LIN {X 0,Y 553.099,Z 303.445,A -85,B 0,C 180,E1 26748.452,E2 26748.452} C_VEL
LIN {X 0,Y 552.954,Z 317.128,A -85,B 0,C 180,E1 26747.901,E2 26747.901} C_VEL
LIN {X 0,Y 552.726,Z 331.261,A -85,B 0,C 180,E1 26747.108,E2 26747.108} C_VEL
LIN {X 0,Y 552.512,Z 344.277,A -85,B 0,C 180,E1 26746.127,E2 26746.127} C_VEL
LIN {X 0,Y 552.313,Z 355.732,A -85,B 0,C 180,E1 26745.002,E2 26745.002} C_VEL
LIN {X 0,Y 552.151,Z 365.084,A -85,B 0,C 180,E1 26743.828,E2 26743.828} C_VEL
LIN {X 0,Y 552.032,Z 373.305,A -85,B 0,C 180,E1 26742.509,E2 26742.509} C_VEL
LIN {X 0,Y 551.958,Z 380.058,A -85,B 0,C 180,E1 26741.069,E2 26741.069} C_VEL
LIN {X 0,Y 551.926,Z 385.3,A -85,B 0,C 180,E1 26739.488,E2 26739.488} C_VEL
LIN {X 0,Y 551.919,Z 388.545,A -85,B 0,C 180,E1 26737.913,E2 26737.913} C_VEL
LIN {X 0,Y 551.917,Z 389.9,A -85,B 0,C 180,E1 26736.448,E2 26736.448} C_VEL
LIN {X 0,Y 551.917,Z 389.555,A -85,B 0,C 180,E1 26734.868,E2 26734.868} C_VEL
LIN {X 0,Y 551.918,Z 387.388,A -85,B 0,C 180,E1 26733.323,E2 26733.323} C_VEL
LIN {X 0,Y 551.933,Z 383.684,A -85,B 0,C 180,E1 26731.868,E2 26731.868} C_VEL
LIN {X 0,Y 551.979,Z 377.809,A -85,B 0,C 180,E1 26730.311,E2 26730.311} C_VEL
LIN {X 0,Y 552.075,Z 370.189,A -85,B 0,C 180,E1 26728.858,E2 26728.858} C_VEL
LIN {X 0,Y 552.222,Z 360.795,A -85,B 0,C 180,E1 26727.509,E2 26727.509} C_VEL
LIN {X 0,Y 552.402,Z 350.546,A -85,B 0,C 180,E1 26726.367,E2 26726.367} C_VEL
LIN {X 0,Y 552.574,Z 339.331,A -85,B 0,C 180,E1 26725.381,E2 26725.381} C_VEL
LIN {X 0,Y 552.815,Z 326.337,A -85,B 0,C 180,E1 26724.499,E2 26724.499} C_VEL
LIN {X 0,Y 552.997,Z 311.82,A -85,B 0,C 180,E1 26723.771,E2 26723.771} C_VEL
LIN {X 0,Y 553.096,Z 297.074,A -85,B 0,C 180,E1 26723.264,E2 26723.264} C_VEL
LIN {X 0,Y 553.162,Z 282.134,A -85,B 0,C 180,E1 26722.957,E2 26722.957} C_VEL
LIN {X 0,Y 553.318,Z 174.705,A -85,B 0,C 180,E1 26721.544,E2 26721.544} C_VEL
LIN {X 0,Y 553.702,Z 126.564,A -85,B 0,C 180,E1 26718.489,E2 26718.489} C_VEL
LIN {X 0,Y 554.116,Z 77.408,A -85,B 0,C 180,E1 26715.367,E2 26715.367} C_VEL
LIN {X 0,Y 554.166,Z 60.38,A -85,B 0,C 180,E1 26714.297,E2 26714.297} C_VEL
LIN {X 0,Y 552.386,Z 53.332,A -85,B 0,C 180,E1 26713.76,E2 26713.76} C_VEL
LIN {X 0,Y 552.341,Z 52.999,A -85,B 0,C 180,E1 26713.258,E2 26713.258} C_VEL
LIN {X 0,Y 552.362,Z 53.27,A -85,B 0,C 180,E1 26712.594,E2 26712.594} C_VEL
LIN {X 0,Y 554.241,Z 59.463,A -85,B 0,C 180,E1 26712.031,E2 26712.031} C_VEL
LIN {X 0,Y 555.025,Z 62.5,A -85,B 0,C 180,E1 26711.786,E2 26711.786} C_VEL
LIN {X 0,Y 554.132,Z 113.525,A -85,B 0,C 180,E1 26708.362,E2 26708.362} C_VEL
LIN {X 0,Y 553.365,Z 164.5,A -85,B 0,C 180,E1 26704.988,E2 26704.988} C_VEL
LIN {X 0,Y 553.381,Z 172.893,A -85,B 0,C 180,E1 26704.473,E2 26704.473} C_VEL
LIN {X 0,Y 553.711,Z 182.776,A -85,B 0,C 180,E1 26704.321,E2 26704.321} C_VEL
LIN {X 0,Y 553.297,Z 287.575,A -85,B 0,C 180,E1 26702.905,E2 26702.905} C_VEL
LIN {X 0,Y 553.196,Z 302.101,A -85,B 0,C 180,E1 26702.529,E2 26702.529} C_VEL
LIN {X 0,Y 553.009,Z 316.307,A -85,B 0,C 180,E1 26701.96,E2 26701.96} C_VEL
LIN {X 0,Y 552.788,Z 329.378,A -85,B 0,C 180,E1 26701.241,E2 26701.241} C_VEL
LIN {X 0,Y 552.561,Z 342.406,A -85,B 0,C 180,E1 26700.293,E2 26700.293} C_VEL
LIN {X 0,Y 552.346,Z 354.092,A -85,B 0,C 180,E1 26699.183,E2 26699.183} C_VEL
LIN {X 0,Y 552.173,Z 363.791,A -85,B 0,C 180,E1 26698.009,E2 26698.009} C_VEL
LIN {X 0,Y 552.049,Z 372.165,A -85,B 0,C 180,E1 26696.716,E2 26696.716} C_VEL
LIN {X 0,Y 551.963,Z 379.488,A -85,B 0,C 180,E1 26695.207,E2 26695.207} C_VEL
LIN {X 0,Y 551.928,Z 384.789,A -85,B 0,C 180,E1 26693.673,E2 26693.673} C_VEL
LIN {X 0,Y 551.918,Z 388.153,A -85,B 0,C 180,E1 26692.173,E2 26692.173} C_VEL
LIN {X 0,Y 551.919,Z 389.809,A -85,B 0,C 180,E1 26690.649,E2 26690.649} C_VEL
LIN {X 0,Y 551.917,Z 389.741,A -85,B 0,C 180,E1 26689.157,E2 26689.157} C_VEL
LIN {X 0,Y 551.918,Z 387.985,A -85,B 0,C 180,E1 26687.63,E2 26687.63} C_VEL
LIN {X 0,Y 551.928,Z 384.27,A -85,B 0,C 180,E1 26686.066,E2 26686.066} C_VEL
LIN {X 0,Y 551.969,Z 379.118,A -85,B 0,C 180,E1 26684.61,E2 26684.61} C_VEL
LIN {X 0,Y 552.051,Z 372.285,A -85,B 0,C 180,E1 26683.206,E2 26683.206} C_VEL
LIN {X 0,Y 552.19,Z 363.437,A -85,B 0,C 180,E1 26681.84,E2 26681.84} C_VEL
LIN {X 0,Y 552.372,Z 353.642,A -85,B 0,C 180,E1 26680.666,E2 26680.666} C_VEL
LIN {X 0,Y 552.577,Z 342.861,A -85,B 0,C 180,E1 26679.641,E2 26679.641} C_VEL
LIN {X 0,Y 552.83,Z 329.763,A -85,B 0,C 180,E1 26678.678,E2 26678.678} C_VEL
LIN {X 0,Y 553.049,Z 316.225,A -85,B 0,C 180,E1 26677.93,E2 26677.93} C_VEL
LIN {X 0,Y 553.237,Z 302.018,A -85,B 0,C 180,E1 26677.362,E2 26677.362} C_VEL
LIN {X 0,Y 553.37,Z 286.424,A -85,B 0,C 180,E1 26676.965,E2 26676.965} C_VEL
LIN {X 0,Y 553.62,Z 179.911,A -85,B 0,C 180,E1 26675.504,E2 26675.504} C_VEL
LIN {X 0,Y 552.92,Z 175.405,A -85,B 0,C 180,E1 26675.389,E2 26675.389} C_VEL
LIN {X 0,Y 553.371,Z 145.57,A -85,B 0,C 180,E1 26672.069,E2 26672.069} C_VEL
LIN {X 0,Y 554.026,Z 115.936,A -85,B 0,C 180,E1 26668.707,E2 26668.707} C_VEL
LIN {X 0,Y 554.696,Z 87.232,A -85,B 0,C 180,E1 26665.405,E2 26665.405} C_VEL
LIN {X 0,Y 555.219,Z 63.854,A -85,B 0,C 180,E1 26662.668,E2 26662.668} C_VEL
LIN {X 0,Y 552.318,Z 53.131,A -85,B 0,C 180,E1 26661.162,E2 26661.162} C_VEL
LIN {X 0,Y 552.344,Z 52.997,A -85,B 0,C 180,E1 26657.923,E2 26657.923} C_VEL
LIN {X 0,Y 552.305,Z 52.997,A -85,B 0,C 180,E1 26654.682,E2 26654.682} C_VEL
LIN {X 0,Y 552.297,Z 52.998,A -85,B 0,C 180,E1 26651.381,E2 26651.381} C_VEL
LIN {X 0,Y 552.344,Z 52.997,A -85,B 0,C 180,E1 26648.117,E2 26648.117} C_VEL
LIN {X 0,Y 552.298,Z 52.998,A -85,B 0,C 180,E1 26644.881,E2 26644.881} C_VEL
LIN {X 0,Y 552.291,Z 52.998,A -85,B 0,C 180,E1 26641.556,E2 26641.556} C_VEL
LIN {X 0,Y 552.345,Z 52.999,A -85,B 0,C 180,E1 26638.341,E2 26638.341} C_VEL
LIN {X 0,Y 552.292,Z 52.998,A -85,B 0,C 180,E1 26635.119,E2 26635.119} C_VEL
LIN {X 0,Y 552.287,Z 52.999,A -85,B 0,C 180,E1 26631.777,E2 26631.777} C_VEL
LIN {X 0,Y 552.34,Z 52.999,A -85,B 0,C 180,E1 26628.514,E2 26628.514} C_VEL
LIN {X 0,Y 552.286,Z 52.998,A -85,B 0,C 180,E1 26625.318,E2 26625.318} C_VEL
LIN {X 0,Y 552.28,Z 52.998,A -85,B 0,C 180,E1 26621.966,E2 26621.966} C_VEL
LIN {X 0,Y 552.342,Z 52.998,A -85,B 0,C 180,E1 26618.774,E2 26618.774} C_VEL
LIN {X 0,Y 552.277,Z 52.999,A -85,B 0,C 180,E1 26615.594,E2 26615.594} C_VEL
LIN {X 0,Y 552.276,Z 53,A -85,B 0,C 180,E1 26612.154,E2 26612.154} C_VEL
LIN {X 0,Y 552.334,Z 53,A -85,B 0,C 180,E1 26608.941,E2 26608.941} C_VEL
LIN {X 0,Y 552.279,Z 53,A -85,B 0,C 180,E1 26605.645,E2 26605.645} C_VEL
LIN {X 0,Y 552.266,Z 53.001,A -85,B 0,C 180,E1 26602.27,E2 26602.27} C_VEL
LIN {X 0,Y 552.323,Z 53.002,A -85,B 0,C 180,E1 26599.056,E2 26599.056} C_VEL
LIN {X 0,Y 552.278,Z 53,A -85,B 0,C 180,E1 26595.812,E2 26595.812} C_VEL
LIN {X 0,Y 552.267,Z 53.002,A -85,B 0,C 180,E1 26592.478,E2 26592.478} C_VEL
LIN {X 0,Y 552.337,Z 52.998,A -85,B 0,C 180,E1 26589.315,E2 26589.315} C_VEL
LIN {X 0,Y 552.282,Z 53.003,A -85,B 0,C 180,E1 26586.043,E2 26586.043} C_VEL
LIN {X 0,Y 552.272,Z 52.996,A -85,B 0,C 180,E1 26582.663,E2 26582.663} C_VEL
LIN {X 0,Y 552.347,Z 53.475,A -85,B 0,C 180,E1 26582.323,E2 26582.323} C_VEL
LIN {X 0,Y 556.547,Z 66.471,A -85,B 0,C 180,E1 26581.038,E2 26581.038} C_VEL
LIN {X 0,Y 555.743,Z 104.341,A -85,B 0,C 180,E1 26578.241,E2 26578.241} C_VEL
LIN {X 0,Y 554.952,Z 151.652,A -85,B 0,C 180,E1 26574.86,E2 26574.86} C_VEL
LIN {X 0,Y 554.938,Z 158.626,A -85,B 0,C 180,E1 26574.402,E2 26574.402} C_VEL
LIN {X 0,Y 555.863,Z 167.052,A -85,B 0,C 180,E1 26574.255,E2 26574.255} C_VEL
LIN {X 0,Y 555.252,Z 366.942,A -85,B 0,C 180,E1 26571.605,E2 26571.605} C_VEL
LIN {X 0,Y 555.016,Z 386.194,A -85,B 0,C 180,E1 26571.154,E2 26571.154} C_VEL
LIN {X 0,Y 554.725,Z 404.372,A -85,B 0,C 180,E1 26570.539,E2 26570.539} C_VEL
LIN {X 0,Y 554.4,Z 421.777,A -85,B 0,C 180,E1 26569.765,E2 26569.765} C_VEL
LIN {X 0,Y 554.022,Z 437.939,A -85,B 0,C 180,E1 26568.848,E2 26568.848} C_VEL
LIN {X 0,Y 553.586,Z 454.217,A -85,B 0,C 180,E1 26567.697,E2 26567.697} C_VEL
LIN {X 0,Y 553.179,Z 468.99,A -85,B 0,C 180,E1 26566.432,E2 26566.432} C_VEL
LIN {X 0,Y 552.81,Z 483.013,A -85,B 0,C 180,E1 26564.99,E2 26564.99} C_VEL
LIN {X 0,Y 552.503,Z 495.909,A -85,B 0,C 180,E1 26563.394,E2 26563.394} C_VEL
LIN {X 0,Y 552.262,Z 507.225,A -85,B 0,C 180,E1 26561.7,E2 26561.7} C_VEL
LIN {X 0,Y 552.098,Z 517.163,A -85,B 0,C 180,E1 26559.872,E2 26559.872} C_VEL
LIN {X 0,Y 551.994,Z 525.176,A -85,B 0,C 180,E1 26558.018,E2 26558.018} C_VEL
LIN {X 0,Y 551.941,Z 531.413,A -85,B 0,C 180,E1 26556.136,E2 26556.136} C_VEL
LIN {X 0,Y 551.914,Z 535.875,A -85,B 0,C 180,E1 26554.26,E2 26554.26} C_VEL
LIN {X 0,Y 551.913,Z 538.792,A -85,B 0,C 180,E1 26552.285,E2 26552.285} C_VEL
LIN {X 0,Y 551.908,Z 539.939,A -85,B 0,C 180,E1 26550.312,E2 26550.312} C_VEL
LIN {X 0,Y 551.913,Z 539.415,A -85,B 0,C 180,E1 26548.444,E2 26548.444} C_VEL
LIN {X 0,Y 551.91,Z 537.163,A -85,B 0,C 180,E1 26546.469,E2 26546.469} C_VEL
LIN {X 0,Y 551.929,Z 533.352,A -85,B 0,C 180,E1 26544.596,E2 26544.596} C_VEL
LIN {X 0,Y 551.964,Z 527.822,A -85,B 0,C 180,E1 26542.716,E2 26542.716} C_VEL
LIN {X 0,Y 552.054,Z 520.43,A -85,B 0,C 180,E1 26540.83,E2 26540.83} C_VEL
LIN {X 0,Y 552.185,Z 511.522,A -85,B 0,C 180,E1 26539.041,E2 26539.041} C_VEL
LIN {X 0,Y 552.389,Z 500.984,A -85,B 0,C 180,E1 26537.323,E2 26537.323} C_VEL
LIN {X 0,Y 552.655,Z 489.359,A -85,B 0,C 180,E1 26535.757,E2 26535.757} C_VEL
LIN {X 0,Y 552.991,Z 476.089,A -85,B 0,C 180,E1 26534.265,E2 26534.265} C_VEL
LIN {X 0,Y 553.394,Z 461.229,A -85,B 0,C 180,E1 26532.873,E2 26532.873} C_VEL
LIN {X 0,Y 553.836,Z 445.249,A -85,B 0,C 180,E1 26531.638,E2 26531.638} C_VEL
LIN {X 0,Y 554.249,Z 428.995,A -85,B 0,C 180,E1 26530.615,E2 26530.615} C_VEL
LIN {X 0,Y 554.606,Z 411.48,A -85,B 0,C 180,E1 26529.75,E2 26529.75} C_VEL
LIN {X 0,Y 554.93,Z 392.522,A -85,B 0,C 180,E1 26529.035,E2 26529.035} C_VEL
LIN {X 0,Y 555.188,Z 373.634,A -85,B 0,C 180,E1 26528.526,E2 26528.526} C_VEL
LIN {X 0,Y 555.342,Z 353.291,A -85,B 0,C 180,E1 26528.186,E2 26528.186} C_VEL
LIN {X 0,Y 555.788,Z 158.707,A -85,B 0,C 180,E1 26525.612,E2 26525.612} C_VEL
LIN {X 0,Y 555.53,Z 154.307,A -85,B 0,C 180,E1 26525.516,E2 26525.516} C_VEL
LIN {X 0,Y 556.369,Z 79.517,A -85,B 0,C 180,E1 26522.378,E2 26522.378} C_VEL
LIN {X 0,Y 556.405,Z 64.239,A -85,B 0,C 180,E1 26521.706,E2 26521.706} C_VEL
LIN {X 0,Y 552.416,Z 53.549,A -85,B 0,C 180,E1 26520.999,E2 26520.999} C_VEL
LIN {X 0,Y 552.331,Z 52.991,A -85,B 0,C 180,E1 26520.755,E2 26520.755} C_VEL
LIN {X 0,Y 552.33,Z 52.994,A -85,B 0,C 180,E1 26517.327,E2 26517.327} C_VEL
LIN {X 0,Y 552.333,Z 52.997,A -85,B 0,C 180,E1 26513.963,E2 26513.963} C_VEL
LIN {X 0,Y 552.342,Z 52.992,A -85,B 0,C 180,E1 26510.553,E2 26510.553} C_VEL
LIN {X 0,Y 552.324,Z 52.995,A -85,B 0,C 180,E1 26507.248,E2 26507.248} C_VEL
LIN {X 0,Y 552.341,Z 52.998,A -85,B 0,C 180,E1 26503.893,E2 26503.893} C_VEL
LIN {X 0,Y 552.336,Z 52.993,A -85,B 0,C 180,E1 26500.512,E2 26500.512} C_VEL
LIN {X 0,Y 552.325,Z 52.993,A -85,B 0,C 180,E1 26497.202,E2 26497.202} C_VEL
LIN {X 0,Y 552.322,Z 52.997,A -85,B 0,C 180,E1 26493.763,E2 26493.763} C_VEL
LIN {X 0,Y 552.339,Z 52.995,A -85,B 0,C 180,E1 26490.455,E2 26490.455} C_VEL
LIN {X 0,Y 552.34,Z 52.99,A -85,B 0,C 180,E1 26487.024,E2 26487.024} C_VEL
LIN {X 0,Y 552.314,Z 52.992,A -85,B 0,C 180,E1 26483.654,E2 26483.654} C_VEL
LIN {X 0,Y 552.335,Z 52.997,A -85,B 0,C 180,E1 26480.335,E2 26480.335} C_VEL
LIN {X 0,Y 552.341,Z 52.994,A -85,B 0,C 180,E1 26476.944,E2 26476.944} C_VEL
LIN {X 0,Y 552.319,Z 52.992,A -85,B 0,C 180,E1 26473.611,E2 26473.611} C_VEL
LIN {X 0,Y 552.313,Z 52.994,A -85,B 0,C 180,E1 26470.219,E2 26470.219} C_VEL
LIN {X 0,Y 552.343,Z 52.998,A -85,B 0,C 180,E1 26466.862,E2 26466.862} C_VEL
LIN {X 0,Y 552.339,Z 52.991,A -85,B 0,C 180,E1 26463.425,E2 26463.425} C_VEL
LIN {X 0,Y 552.306,Z 52.992,A -85,B 0,C 180,E1 26460.104,E2 26460.104} C_VEL
LIN {X 0,Y 552.323,Z 52.998,A -85,B 0,C 180,E1 26456.762,E2 26456.762} C_VEL
LIN {X 0,Y 552.344,Z 52.993,A -85,B 0,C 180,E1 26453.451,E2 26453.451} C_VEL
LIN {X 0,Y 552.304,Z 52.993,A -85,B 0,C 180,E1 26450.202,E2 26450.202} C_VEL
LIN {X 0,Y 552.31,Z 52.995,A -85,B 0,C 180,E1 26446.814,E2 26446.814} C_VEL
LIN {X 0,Y 552.344,Z 52.997,A -85,B 0,C 180,E1 26443.489,E2 26443.489} C_VEL
LIN {X 0,Y 552.31,Z 52.995,A -85,B 0,C 180,E1 26440.212,E2 26440.212} C_VEL
LIN {X 0,Y 552.298,Z 52.989,A -85,B 0,C 180,E1 26436.868,E2 26436.868} C_VEL
LIN {X 0,Y 552.341,Z 52.998,A -85,B 0,C 180,E1 26433.556,E2 26433.556} C_VEL
LIN {X 0,Y 552.294,Z 52.997,A -85,B 0,C 180,E1 26432.704,E2 26432.704} C_VEL
LIN {X 0,Y 551.318,Z 53.124,A -85,B 0,C 180,E1 26431.905,E2 26431.905} C_VEL
LIN {X 0,Y 544.811,Z 53.932,A -85,B 0,C 180,E1 26429.603,E2 26429.603} C_VEL
LIN {X 0,Y 544.359,Z 53.984,A -85,B 0,C 180,E1 26429.076,E2 26429.076} C_VEL
LIN {X 0,Y 544.403,Z 53.986,A -85,B 0,C 180,E1 26425.736,E2 26425.736} C_VEL
LIN {X 0,Y 544.373,Z 53.985,A -85,B 0,C 180,E1 26422.425,E2 26422.425} C_VEL
LIN {X 0,Y 544.352,Z 53.986,A -85,B 0,C 180,E1 26419.164,E2 26419.164} C_VEL
LIN {X 0,Y 544.395,Z 53.985,A -85,B 0,C 180,E1 26415.886,E2 26415.886} C_VEL
LIN {X 0,Y 544.364,Z 53.983,A -85,B 0,C 180,E1 26412.667,E2 26412.667} C_VEL
LIN {X 0,Y 544.344,Z 53.99,A -85,B 0,C 180,E1 26409.322,E2 26409.322} C_VEL
LIN {X 0,Y 544.391,Z 53.989,A -85,B 0,C 180,E1 26406.086,E2 26406.086} C_VEL
LIN {X 0,Y 544.387,Z 54.212,A -85,B 0,C 180,E1 26403.766,E2 26403.766} C_VEL
LIN {X 0,Y 545.826,Z 61.376,A -85,B 0,C 180,E1 26402.958,E2 26402.958} C_VEL
LIN {X 0,Y 545.926,Z 92.268,A -85,B 0,C 180,E1 26399.756,E2 26399.756} C_VEL
LIN {X 0,Y 545.776,Z 123.082,A -85,B 0,C 180,E1 26396.489,E2 26396.489} C_VEL
LIN {X 0,Y 545.516,Z 153.208,A -85,B 0,C 180,E1 26393.264,E2 26393.264} C_VEL
LIN {X 0,Y 545.269,Z 178.791,A -85,B 0,C 180,E1 26390.544,E2 26390.544} C_VEL
LIN {X 0,Y 545.789,Z 185.113,A -85,B 0,C 180,E1 26390.438,E2 26390.438} C_VEL
LIN {X 0,Y 545.419,Z 289.991,A -85,B 0,C 180,E1 26389.023,E2 26389.023} C_VEL
LIN {X 0,Y 545.341,Z 304.564,A -85,B 0,C 180,E1 26388.63,E2 26388.63} C_VEL
LIN {X 0,Y 545.187,Z 318.586,A -85,B 0,C 180,E1 26388.055,E2 26388.055} C_VEL
LIN {X 0,Y 544.956,Z 332.024,A -85,B 0,C 180,E1 26387.29,E2 26387.29} C_VEL
LIN {X 0,Y 544.717,Z 344.949,A -85,B 0,C 180,E1 26386.309,E2 26386.309} C_VEL
LIN {X 0,Y 544.502,Z 356.015,A -85,B 0,C 180,E1 26385.223,E2 26385.223} C_VEL
LIN {X 0,Y 544.314,Z 365.564,A -85,B 0,C 180,E1 26384.031,E2 26384.031} C_VEL
LIN {X 0,Y 544.159,Z 374.274,A -85,B 0,C 180,E1 26382.629,E2 26382.629} C_VEL
LIN {X 0,Y 544.062,Z 381.231,A -85,B 0,C 180,E1 26381.125,E2 26381.125} C_VEL
LIN {X 0,Y 544.009,Z 386.403,A -85,B 0,C 180,E1 26379.52,E2 26379.52} C_VEL
LIN {X 0,Y 543.982,Z 389.541,A -85,B 0,C 180,E1 26377.923,E2 26377.923} C_VEL
LIN {X 0,Y 543.971,Z 390.853,A -85,B 0,C 180,E1 26376.331,E2 26376.331} C_VEL
LIN {X 0,Y 543.973,Z 390.407,A -85,B 0,C 180,E1 26374.744,E2 26374.744} C_VEL
LIN {X 0,Y 543.991,Z 387.95,A -85,B 0,C 180,E1 26373.055,E2 26373.055} C_VEL
LIN {X 0,Y 544.033,Z 383.689,A -85,B 0,C 180,E1 26371.474,E2 26371.474} C_VEL
LIN {X 0,Y 544.102,Z 377.829,A -85,B 0,C 180,E1 26369.999,E2 26369.999} C_VEL
LIN {X 0,Y 544.219,Z 370.506,A -85,B 0,C 180,E1 26368.631,E2 26368.631} C_VEL
LIN {X 0,Y 544.385,Z 361.73,A -85,B 0,C 180,E1 26367.367,E2 26367.367} C_VEL
LIN {X 0,Y 544.591,Z 351.43,A -85,B 0,C 180,E1 26366.21,E2 26366.21} C_VEL
LIN {X 0,Y 544.785,Z 340.151,A -85,B 0,C 180,E1 26365.209,E2 26365.209} C_VEL
LIN {X 0,Y 545.047,Z 327.077,A -85,B 0,C 180,E1 26364.314,E2 26364.314} C_VEL
LIN {X 0,Y 545.241,Z 312.435,A -85,B 0,C 180,E1 26363.577,E2 26363.577} C_VEL
LIN {X 0,Y 545.348,Z 296.996,A -85,B 0,C 180,E1 26363.049,E2 26363.049} C_VEL
LIN {X 0,Y 545.398,Z 281.169,A -85,B 0,C 180,E1 26362.742,E2 26362.742} C_VEL
LIN {X 0,Y 545.609,Z 175.423,A -85,B 0,C 180,E1 26361.33,E2 26361.33} C_VEL
LIN {X 0,Y 546.063,Z 123.971,A -85,B 0,C 180,E1 26358.058,E2 26358.058} C_VEL
LIN {X 0,Y 546.484,Z 71.6,A -85,B 0,C 180,E1 26354.724,E2 26354.724} C_VEL
LIN {X 0,Y 546.407,Z 61.981,A -85,B 0,C 180,E1 26354.123,E2 26354.123} C_VEL
LIN {X 0,Y 544.455,Z 54.321,A -85,B 0,C 180,E1 26353.53,E2 26353.53} C_VEL
LIN {X 0,Y 544.396,Z 53.991,A -85,B 0,C 180,E1 26353.116,E2 26353.116} C_VEL
LIN {X 0,Y 544.488,Z 54.61,A -85,B 0,C 180,E1 26352.858,E2 26352.858} C_VEL
LIN {X 0,Y 547.518,Z 64.97,A -85,B 0,C 180,E1 26351.968,E2 26351.968} C_VEL
LIN {X 0,Y 546.527,Z 115.573,A -85,B 0,C 180,E1 26348.537,E2 26348.537} C_VEL
LIN {X 0,Y 545.66,Z 166.93,A -85,B 0,C 180,E1 26345.099,E2 26345.099} C_VEL
LIN {X 0,Y 545.704,Z 172.937,A -85,B 0,C 180,E1 26344.742,E2 26344.742} C_VEL
LIN {X 0,Y 546.13,Z 181.831,A -85,B 0,C 180,E1 26344.6,E2 26344.6} C_VEL
LIN {X 0,Y 545.622,Z 288.062,A -85,B 0,C 180,E1 26343.135,E2 26343.135} C_VEL
LIN {X 0,Y 545.499,Z 303.41,A -85,B 0,C 180,E1 26342.727,E2 26342.727} C_VEL
LIN {X 0,Y 545.278,Z 318.268,A -85,B 0,C 180,E1 26342.109,E2 26342.109} C_VEL
LIN {X 0,Y 545.031,Z 330.81,A -85,B 0,C 180,E1 26341.392,E2 26341.392} C_VEL
LIN {X 0,Y 544.781,Z 343.449,A -85,B 0,C 180,E1 26340.454,E2 26340.454} C_VEL
LIN {X 0,Y 544.529,Z 355.341,A -85,B 0,C 180,E1 26339.305,E2 26339.305} C_VEL
LIN {X 0,Y 544.324,Z 365.014,A -85,B 0,C 180,E1 26338.108,E2 26338.108} C_VEL
LIN {X 0,Y 544.175,Z 373.324,A -85,B 0,C 180,E1 26336.801,E2 26336.801} C_VEL
LIN {X 0,Y 544.066,Z 380.786,A -85,B 0,C 180,E1 26335.233,E2 26335.233} C_VEL
LIN {X 0,Y 544.01,Z 386.15,A -85,B 0,C 180,E1 26333.613,E2 26333.613} C_VEL
LIN {X 0,Y 543.982,Z 389.363,A -85,B 0,C 180,E1 26332.048,E2 26332.048} C_VEL
LIN {X 0,Y 543.973,Z 390.829,A -85,B 0,C 180,E1 26330.508,E2 26330.508} C_VEL
LIN {X 0,Y 543.975,Z 390.517,A -85,B 0,C 180,E1 26328.85,E2 26328.85} C_VEL
LIN {X 0,Y 543.995,Z 388.455,A -85,B 0,C 180,E1 26327.295,E2 26327.295} C_VEL
LIN {X 0,Y 544.035,Z 384.784,A -85,B 0,C 180,E1 26325.788,E2 26325.788} C_VEL
LIN {X 0,Y 544.105,Z 378.968,A -85,B 0,C 180,E1 26324.22,E2 26324.22} C_VEL
LIN {X 0,Y 544.222,Z 371.846,A -85,B 0,C 180,E1 26322.826,E2 26322.826} C_VEL
LIN {X 0,Y 544.398,Z 363.265,A -85,B 0,C 180,E1 26321.531,E2 26321.531} C_VEL
LIN {X 0,Y 544.642,Z 352.354,A -85,B 0,C 180,E1 26320.257,E2 26320.257} C_VEL
LIN {X 0,Y 544.89,Z 340.946,A -85,B 0,C 180,E1 26319.222,E2 26319.222} C_VEL
LIN {X 0,Y 545.16,Z 328.543,A -85,B 0,C 180,E1 26318.343,E2 26318.343} C_VEL
LIN {X 0,Y 545.405,Z 315.197,A -85,B 0,C 180,E1 26317.624,E2 26317.624} C_VEL
LIN {X 0,Y 545.601,Z 300.554,A -85,B 0,C 180,E1 26317.062,E2 26317.062} C_VEL
LIN {X 0,Y 545.735,Z 285.71,A -85,B 0,C 180,E1 26316.702,E2 26316.702} C_VEL
LIN {X 0,Y 546.094,Z 180.817,A -85,B 0,C 180,E1 26315.23,E2 26315.23} C_VEL
LIN {X 0,Y 545.172,Z 175.182,A -85,B 0,C 180,E1 26315.082,E2 26315.082} C_VEL
LIN {X 0,Y 545.69,Z 145.44,A -85,B 0,C 180,E1 26311.727,E2 26311.727} C_VEL
LIN {X 0,Y 546.426,Z 115.516,A -85,B 0,C 180,E1 26308.29,E2 26308.29} C_VEL
LIN {X 0,Y 547.207,Z 87.033,A -85,B 0,C 180,E1 26304.967,E2 26304.967} C_VEL
LIN {X 0,Y 547.749,Z 66.487,A -85,B 0,C 180,E1 26302.535,E2 26302.535} C_VEL
LIN {X 0,Y 544.375,Z 54.101,A -85,B 0,C 180,E1 26300.762,E2 26300.762} C_VEL
LIN {X 0,Y 544.369,Z 53.99,A -85,B 0,C 180,E1 26297.421,E2 26297.421} C_VEL
LIN {X 0,Y 544.409,Z 53.986,A -85,B 0,C 180,E1 26294.136,E2 26294.136} C_VEL
LIN {X 0,Y 544.356,Z 53.986,A -85,B 0,C 180,E1 26290.906,E2 26290.906} C_VEL
LIN {X 0,Y 544.356,Z 53.988,A -85,B 0,C 180,E1 26287.494,E2 26287.494} C_VEL
LIN {X 0,Y 544.404,Z 53.988,A -85,B 0,C 180,E1 26284.213,E2 26284.213} C_VEL
LIN {X 0,Y 544.36,Z 53.986,A -85,B 0,C 180,E1 26280.947,E2 26280.947} C_VEL
LIN {X 0,Y 544.347,Z 53.988,A -85,B 0,C 180,E1 26277.579,E2 26277.579} C_VEL
LIN {X 0,Y 544.397,Z 53.988,A -85,B 0,C 180,E1 26274.308,E2 26274.308} C_VEL
LIN {X 0,Y 544.357,Z 53.987,A -85,B 0,C 180,E1 26271.125,E2 26271.125} C_VEL
LIN {X 0,Y 544.343,Z 53.988,A -85,B 0,C 180,E1 26267.737,E2 26267.737} C_VEL
LIN {X 0,Y 544.386,Z 53.988,A -85,B 0,C 180,E1 26264.446,E2 26264.446} C_VEL
LIN {X 0,Y 544.355,Z 53.986,A -85,B 0,C 180,E1 26261.25,E2 26261.25} C_VEL
LIN {X 0,Y 544.337,Z 53.988,A -85,B 0,C 180,E1 26257.993,E2 26257.993} C_VEL
LIN {X 0,Y 544.394,Z 53.989,A -85,B 0,C 180,E1 26254.78,E2 26254.78} C_VEL
LIN {X 0,Y 544.341,Z 53.989,A -85,B 0,C 180,E1 26251.593,E2 26251.593} C_VEL
LIN {X 0,Y 544.331,Z 53.99,A -85,B 0,C 180,E1 26248.185,E2 26248.185} C_VEL
LIN {X 0,Y 544.383,Z 53.99,A -85,B 0,C 180,E1 26244.909,E2 26244.909} C_VEL
LIN {X 0,Y 544.342,Z 53.99,A -85,B 0,C 180,E1 26241.658,E2 26241.658} C_VEL
LIN {X 0,Y 544.324,Z 53.991,A -85,B 0,C 180,E1 26238.322,E2 26238.322} C_VEL
LIN {X 0,Y 544.386,Z 53.989,A -85,B 0,C 180,E1 26235.148,E2 26235.148} C_VEL
LIN {X 0,Y 544.34,Z 53.991,A -85,B 0,C 180,E1 26231.934,E2 26231.934} C_VEL
LIN {X 0,Y 544.334,Z 53.992,A -85,B 0,C 180,E1 26228.648,E2 26228.648} C_VEL
LIN {X 0,Y 544.392,Z 53.989,A -85,B 0,C 180,E1 26225.366,E2 26225.366} C_VEL
LIN {X 0,Y 544.376,Z 54.248,A -85,B 0,C 180,E1 26222.777,E2 26222.777} C_VEL
LIN {X 0,Y 549.194,Z 68.607,A -85,B 0,C 180,E1 26221.293,E2 26221.293} C_VEL
LIN {X 0,Y 548.134,Z 110.619,A -85,B 0,C 180,E1 26218.134,E2 26218.134} C_VEL
LIN {X 0,Y 547.224,Z 157.206,A -85,B 0,C 180,E1 26214.757,E2 26214.757} C_VEL
LIN {X 0,Y 547.437,Z 159.937,A -85,B 0,C 180,E1 26214.657,E2 26214.657} C_VEL
LIN {X 0,Y 548.298,Z 168.095,A -85,B 0,C 180,E1 26214.515,E2 26214.515} C_VEL
LIN {X 0,Y 547.592,Z 366.306,A -85,B 0,C 180,E1 26211.855,E2 26211.855} C_VEL
LIN {X 0,Y 547.319,Z 385.448,A -85,B 0,C 180,E1 26211.402,E2 26211.402} C_VEL
LIN {X 0,Y 546.977,Z 403.863,A -85,B 0,C 180,E1 26210.771,E2 26210.771} C_VEL
LIN {X 0,Y 546.58,Z 422.045,A -85,B 0,C 180,E1 26209.943,E2 26209.943} C_VEL
LIN {X 0,Y 546.163,Z 439.093,A -85,B 0,C 180,E1 26208.963,E2 26208.963} C_VEL
LIN {X 0,Y 545.743,Z 455.363,A -85,B 0,C 180,E1 26207.817,E2 26207.817} C_VEL
LIN {X 0,Y 545.352,Z 470.045,A -85,B 0,C 180,E1 26206.565,E2 26206.565} C_VEL
LIN {X 0,Y 544.957,Z 483.221,A -85,B 0,C 180,E1 26205.187,E2 26205.187} C_VEL
LIN {X 0,Y 544.604,Z 495.908,A -85,B 0,C 180,E1 26203.592,E2 26203.592} C_VEL
LIN {X 0,Y 544.327,Z 507.224,A -85,B 0,C 180,E1 26201.873,E2 26201.873} C_VEL
LIN {X 0,Y 544.133,Z 516.989,A -85,B 0,C 180,E1 26200.054,E2 26200.054} C_VEL
LIN {X 0,Y 544.007,Z 525.175,A -85,B 0,C 180,E1 26198.137,E2 26198.137} C_VEL
LIN {X 0,Y 543.944,Z 531.413,A -85,B 0,C 180,E1 26196.227,E2 26196.227} C_VEL
LIN {X 0,Y 543.916,Z 535.875,A -85,B 0,C 180,E1 26194.323,E2 26194.323} C_VEL
LIN {X 0,Y 543.912,Z 538.791,A -85,B 0,C 180,E1 26192.319,E2 26192.319} C_VEL
LIN {X 0,Y 543.908,Z 539.939,A -85,B 0,C 180,E1 26190.317,E2 26190.317} C_VEL
LIN {X 0,Y 543.912,Z 539.415,A -85,B 0,C 180,E1 26188.421,E2 26188.421} C_VEL
LIN {X 0,Y 543.911,Z 537.162,A -85,B 0,C 180,E1 26186.417,E2 26186.417} C_VEL
LIN {X 0,Y 543.931,Z 533.351,A -85,B 0,C 180,E1 26184.516,E2 26184.516} C_VEL
LIN {X 0,Y 543.976,Z 527.821,A -85,B 0,C 180,E1 26182.609,E2 26182.609} C_VEL
LIN {X 0,Y 544.076,Z 520.43,A -85,B 0,C 180,E1 26180.694,E2 26180.694} C_VEL
LIN {X 0,Y 544.236,Z 511.522,A -85,B 0,C 180,E1 26178.879,E2 26178.879} C_VEL
LIN {X 0,Y 544.467,Z 501.156,A -85,B 0,C 180,E1 26177.163,E2 26177.163} C_VEL
LIN {X 0,Y 544.783,Z 489.358,A -85,B 0,C 180,E1 26175.547,E2 26175.547} C_VEL
LIN {X 0,Y 545.177,Z 476.088,A -85,B 0,C 180,E1 26174.033,E2 26174.033} C_VEL
LIN {X 0,Y 545.549,Z 462.781,A -85,B 0,C 180,E1 26172.784,E2 26172.784} C_VEL
LIN {X 0,Y 545.973,Z 446.914,A -85,B 0,C 180,E1 26171.556,E2 26171.556} C_VEL
LIN {X 0,Y 546.404,Z 430.208,A -85,B 0,C 180,E1 26170.492,E2 26170.492} C_VEL
LIN {X 0,Y 546.805,Z 413.145,A -85,B 0,C 180,E1 26169.616,E2 26169.616} C_VEL
LIN {X 0,Y 547.176,Z 395.356,A -85,B 0,C 180,E1 26168.902,E2 26168.902} C_VEL
LIN {X 0,Y 547.488,Z 376.64,A -85,B 0,C 180,E1 26168.353,E2 26168.353} C_VEL
LIN {X 0,Y 547.698,Z 357.218,A -85,B 0,C 180,E1 26167.987,E2 26167.987} C_VEL
LIN {X 0,Y 548.265,Z 159.461,A -85,B 0,C 180,E1 26165.338,E2 26165.338} C_VEL
LIN {X 0,Y 547.969,Z 154.53,A -85,B 0,C 180,E1 26165.236,E2 26165.236} C_VEL
LIN {X 0,Y 548.899,Z 86.989,A -85,B 0,C 180,E1 26162.353,E2 26162.353} C_VEL
LIN {X 0,Y 549.159,Z 66.994,A -85,B 0,C 180,E1 26161.472,E2 26161.472} C_VEL
LIN {X 0,Y 544.495,Z 54.583,A -85,B 0,C 180,E1 26160.642,E2 26160.642} C_VEL
LIN {X 0,Y 544.41,Z 54.031,A -85,B 0,C 180,E1 26160.516,E2 26160.516} C_VEL
LIN {X 0,Y 544.387,Z 53.981,A -85,B 0,C 180,E1 26157.069,E2 26157.069} C_VEL
LIN {X 0,Y 544.4,Z 53.988,A -85,B 0,C 180,E1 26153.734,E2 26153.734} C_VEL
LIN {X 0,Y 544.394,Z 53.985,A -85,B 0,C 180,E1 26150.273,E2 26150.273} C_VEL
LIN {X 0,Y 544.395,Z 53.982,A -85,B 0,C 180,E1 26146.905,E2 26146.905} C_VEL
LIN {X 0,Y 544.385,Z 53.985,A -85,B 0,C 180,E1 26143.493,E2 26143.493} C_VEL
LIN {X 0,Y 544.401,Z 53.986,A -85,B 0,C 180,E1 26140.14,E2 26140.14} C_VEL
LIN {X 0,Y 544.399,Z 53.982,A -85,B 0,C 180,E1 26136.648,E2 26136.648} C_VEL
LIN {X 0,Y 544.385,Z 53.982,A -85,B 0,C 180,E1 26133.31,E2 26133.31} C_VEL
LIN {X 0,Y 544.383,Z 53.986,A -85,B 0,C 180,E1 26129.851,E2 26129.851} C_VEL
LIN {X 0,Y 544.4,Z 53.984,A -85,B 0,C 180,E1 26126.506,E2 26126.506} C_VEL
LIN {X 0,Y 544.404,Z 53.977,A -85,B 0,C 180,E1 26123.029,E2 26123.029} C_VEL
LIN {X 0,Y 544.375,Z 53.981,A -85,B 0,C 180,E1 26119.64,E2 26119.64} C_VEL
LIN {X 0,Y 544.382,Z 53.986,A -85,B 0,C 180,E1 26116.211,E2 26116.211} C_VEL
LIN {X 0,Y 544.401,Z 53.984,A -85,B 0,C 180,E1 26112.84,E2 26112.84} C_VEL
LIN {X 0,Y 544.397,Z 53.978,A -85,B 0,C 180,E1 26109.408,E2 26109.408} C_VEL
LIN {X 0,Y 544.369,Z 53.984,A -85,B 0,C 180,E1 26106.115,E2 26106.115} C_VEL
LIN {X 0,Y 544.392,Z 53.988,A -85,B 0,C 180,E1 26102.737,E2 26102.737} C_VEL
LIN {X 0,Y 544.406,Z 53.979,A -85,B 0,C 180,E1 26099.368,E2 26099.368} C_VEL
LIN {X 0,Y 544.372,Z 53.982,A -85,B 0,C 180,E1 26095.998,E2 26095.998} C_VEL
LIN {X 0,Y 544.371,Z 53.986,A -85,B 0,C 180,E1 26092.613,E2 26092.613} C_VEL
LIN {X 0,Y 544.403,Z 53.984,A -85,B 0,C 180,E1 26089.283,E2 26089.283} C_VEL
LIN {X 0,Y 544.392,Z 53.979,A -85,B 0,C 180,E1 26085.864,E2 26085.864} C_VEL
LIN {X 0,Y 544.36,Z 53.983,A -85,B 0,C 180,E1 26082.579,E2 26082.579} C_VEL
LIN {X 0,Y 544.385,Z 53.986,A -85,B 0,C 180,E1 26079.202,E2 26079.202} C_VEL
LIN {X 0,Y 544.403,Z 53.974,A -85,B 0,C 180,E1 26075.822,E2 26075.822} C_VEL
LIN {X 0,Y 544.36,Z 53.985,A -85,B 0,C 180,E1 26072.514,E2 26072.514} C_VEL
LIN {X 0,Y 544.359,Z 53.984,A -85,B 0,C 180,E1 26069.076,E2 26069.076} C_VEL
LIN {X 0,Y 543.365,Z 54.108,A -85,B 0,C 180,E1 26068.266,E2 26068.266} C_VEL
LIN {X 0,Y 536.893,Z 54.923,A -85,B 0,C 180,E1 26065.929,E2 26065.929} C_VEL
LIN {X 0,Y 536.432,Z 54.972,A -85,B 0,C 180,E1 26065.395,E2 26065.395} C_VEL
LIN {X 0,Y 536.468,Z 54.974,A -85,B 0,C 180,E1 26062.032,E2 26062.032} C_VEL
LIN {X 0,Y 536.419,Z 54.974,A -85,B 0,C 180,E1 26058.69,E2 26058.69} C_VEL
LIN {X 0,Y 536.412,Z 54.977,A -85,B 0,C 180,E1 26055.354,E2 26055.354} C_VEL
LIN {X 0,Y 536.465,Z 54.974,A -85,B 0,C 180,E1 26052.115,E2 26052.115} C_VEL
LIN {X 0,Y 536.419,Z 54.978,A -85,B 0,C 180,E1 26048.818,E2 26048.818} C_VEL
LIN {X 0,Y 536.406,Z 54.982,A -85,B 0,C 180,E1 26045.428,E2 26045.428} C_VEL
LIN {X 0,Y 536.469,Z 55.193,A -85,B 0,C 180,E1 26044.01,E2 26044.01} C_VEL
LIN {X 0,Y 538.146,Z 63.457,A -85,B 0,C 180,E1 26043.076,E2 26043.076} C_VEL
LIN {X 0,Y 538.214,Z 93.891,A -85,B 0,C 180,E1 26039.903,E2 26039.903} C_VEL
LIN {X 0,Y 538.036,Z 124.559,A -85,B 0,C 180,E1 26036.636,E2 26036.636} C_VEL
LIN {X 0,Y 537.755,Z 155.816,A -85,B 0,C 180,E1 26033.291,E2 26033.291} C_VEL
LIN {X 0,Y 537.539,Z 179.646,A -85,B 0,C 180,E1 26030.762,E2 26030.762} C_VEL
LIN {X 0,Y 538.072,Z 185.697,A -85,B 0,C 180,E1 26030.656,E2 26030.656} C_VEL
LIN {X 0,Y 537.665,Z 291.177,A -85,B 0,C 180,E1 26029.211,E2 26029.211} C_VEL
LIN {X 0,Y 537.59,Z 305.539,A -85,B 0,C 180,E1 26028.819,E2 26028.819} C_VEL
LIN {X 0,Y 537.437,Z 319.291,A -85,B 0,C 180,E1 26028.251,E2 26028.251} C_VEL
LIN {X 0,Y 537.177,Z 333.403,A -85,B 0,C 180,E1 26027.437,E2 26027.437} C_VEL
LIN {X 0,Y 536.92,Z 346.267,A -85,B 0,C 180,E1 26026.442,E2 26026.442} C_VEL
LIN {X 0,Y 536.678,Z 357.282,A -85,B 0,C 180,E1 26025.339,E2 26025.339} C_VEL
LIN {X 0,Y 536.464,Z 366.793,A -85,B 0,C 180,E1 26024.131,E2 26024.131} C_VEL
LIN {X 0,Y 536.297,Z 374.89,A -85,B 0,C 180,E1 26022.817,E2 26022.817} C_VEL
LIN {X 0,Y 536.173,Z 381.966,A -85,B 0,C 180,E1 26021.291,E2 26021.291} C_VEL
LIN {X 0,Y 536.103,Z 386.969,A -85,B 0,C 180,E1 26019.771,E2 26019.771} C_VEL
LIN {X 0,Y 536.066,Z 390.205,A -85,B 0,C 180,E1 26018.256,E2 26018.256} C_VEL
LIN {X 0,Y 536.049,Z 391.905,A -85,B 0,C 180,E1 26016.532,E2 26016.532} C_VEL
LIN {X 0,Y 536.049,Z 391.568,A -85,B 0,C 180,E1 26014.814,E2 26014.814} C_VEL
LIN {X 0,Y 536.069,Z 389.401,A -85,B 0,C 180,E1 26013.207,E2 26013.207} C_VEL
LIN {X 0,Y 536.118,Z 385.723,A -85,B 0,C 180,E1 26011.709,E2 26011.709} C_VEL
LIN {X 0,Y 536.196,Z 380.278,A -85,B 0,C 180,E1 26010.213,E2 26010.213} C_VEL
LIN {X 0,Y 536.332,Z 372.741,A -85,B 0,C 180,E1 26008.717,E2 26008.717} C_VEL
LIN {X 0,Y 536.512,Z 364.265,A -85,B 0,C 180,E1 26007.436,E2 26007.436} C_VEL
LIN {X 0,Y 536.738,Z 354.405,A -85,B 0,C 180,E1 26006.261,E2 26006.261} C_VEL
LIN {X 0,Y 536.98,Z 342.336,A -85,B 0,C 180,E1 26005.139,E2 26005.139} C_VEL
LIN {X 0,Y 537.244,Z 329.557,A -85,B 0,C 180,E1 26004.231,E2 26004.231} C_VEL
LIN {X 0,Y 537.455,Z 316.607,A -85,B 0,C 180,E1 26003.537,E2 26003.537} C_VEL
LIN {X 0,Y 537.567,Z 302.3,A -85,B 0,C 180,E1 26002.985,E2 26002.985} C_VEL
LIN {X 0,Y 537.632,Z 286.721,A -85,B 0,C 180,E1 26002.615,E2 26002.615} C_VEL
LIN {X 0,Y 537.903,Z 176.124,A -85,B 0,C 180,E1 26001.111,E2 26001.111} C_VEL
LIN {X 0,Y 538.401,Z 123.883,A -85,B 0,C 180,E1 25997.777,E2 25997.777} C_VEL
LIN {X 0,Y 538.82,Z 72.538,A -85,B 0,C 180,E1 25994.501,E2 25994.501} C_VEL
LIN {X 0,Y 538.728,Z 63.801,A -85,B 0,C 180,E1 25993.946,E2 25993.946} C_VEL
LIN {X 0,Y 536.715,Z 56.195,A -85,B 0,C 180,E1 25993.355,E2 25993.355} C_VEL
LIN {X 0,Y 536.654,Z 55.991,A -85,B 0,C 180,E1 25993.186,E2 25993.186} C_VEL
LIN {X 0,Y 538.216,Z 60.929,A -85,B 0,C 180,E1 25992.708,E2 25992.708} C_VEL
LIN {X 0,Y 540.022,Z 67.463,A -85,B 0,C 180,E1 25992.155,E2 25992.155} C_VEL
LIN {X 0,Y 538.909,Z 118.57,A -85,B 0,C 180,E1 25988.652,E2 25988.652} C_VEL
LIN {X 0,Y 537.946,Z 170.132,A -85,B 0,C 180,E1 25985.161,E2 25985.161} C_VEL
LIN {X 0,Y 538.064,Z 173.179,A -85,B 0,C 180,E1 25985.017,E2 25985.017} C_VEL
LIN {X 0,Y 538.556,Z 181.813,A -85,B 0,C 180,E1 25984.874,E2 25984.874} C_VEL
LIN {X 0,Y 537.954,Z 288.762,A -85,B 0,C 180,E1 25983.366,E2 25983.366} C_VEL
LIN {X 0,Y 537.818,Z 303.711,A -85,B 0,C 180,E1 25982.964,E2 25982.964} C_VEL
LIN {X 0,Y 537.579,Z 318.393,A -85,B 0,C 180,E1 25982.351,E2 25982.351} C_VEL
LIN {X 0,Y 537.305,Z 331.227,A -85,B 0,C 180,E1 25981.617,E2 25981.617} C_VEL
LIN {X 0,Y 537.02,Z 343.771,A -85,B 0,C 180,E1 25980.681,E2 25980.681} C_VEL
LIN {X 0,Y 536.739,Z 355.419,A -85,B 0,C 180,E1 25979.556,E2 25979.556} C_VEL
LIN {X 0,Y 536.51,Z 364.934,A -85,B 0,C 180,E1 25978.396,E2 25978.396} C_VEL
LIN {X 0,Y 536.318,Z 373.77,A -85,B 0,C 180,E1 25977.018,E2 25977.018} C_VEL
LIN {X 0,Y 536.186,Z 380.677,A -85,B 0,C 180,E1 25975.596,E2 25975.596} C_VEL
LIN {X 0,Y 536.118,Z 385.884,A -85,B 0,C 180,E1 25974.154,E2 25974.154} C_VEL
LIN {X 0,Y 536.068,Z 389.911,A -85,B 0,C 180,E1 25972.439,E2 25972.439} C_VEL
LIN {X 0,Y 536.051,Z 391.783,A -85,B 0,C 180,E1 25970.779,E2 25970.779} C_VEL
LIN {X 0,Y 536.055,Z 391.874,A -85,B 0,C 180,E1 25969.225,E2 25969.225} C_VEL
LIN {X 0,Y 536.078,Z 390.095,A -85,B 0,C 180,E1 25967.532,E2 25967.532} C_VEL
LIN {X 0,Y 536.128,Z 386.398,A -85,B 0,C 180,E1 25965.891,E2 25965.891} C_VEL
LIN {X 0,Y 536.213,Z 381.101,A -85,B 0,C 180,E1 25964.367,E2 25964.367} C_VEL
LIN {X 0,Y 536.355,Z 374.036,A -85,B 0,C 180,E1 25962.893,E2 25962.893} C_VEL
LIN {X 0,Y 536.566,Z 365.089,A -85,B 0,C 180,E1 25961.487,E2 25961.487} C_VEL
LIN {X 0,Y 536.822,Z 355.024,A -85,B 0,C 180,E1 25960.264,E2 25960.264} C_VEL
LIN {X 0,Y 537.1,Z 344.128,A -85,B 0,C 180,E1 25959.214,E2 25959.214} C_VEL
LIN {X 0,Y 537.429,Z 330.961,A -85,B 0,C 180,E1 25958.229,E2 25958.229} C_VEL
LIN {X 0,Y 537.718,Z 316.868,A -85,B 0,C 180,E1 25957.441,E2 25957.441} C_VEL
LIN {X 0,Y 537.941,Z 302.692,A -85,B 0,C 180,E1 25956.871,E2 25956.871} C_VEL
LIN {X 0,Y 538.096,Z 287.502,A -85,B 0,C 180,E1 25956.476,E2 25956.476} C_VEL
LIN {X 0,Y 538.591,Z 181.923,A -85,B 0,C 180,E1 25954.952,E2 25954.952} C_VEL
LIN {X 0,Y 537.435,Z 175.11,A -85,B 0,C 180,E1 25954.778,E2 25954.778} C_VEL
LIN {X 0,Y 538.014,Z 146.054,A -85,B 0,C 180,E1 25951.459,E2 25951.459} C_VEL
LIN {X 0,Y 538.846,Z 116.045,A -85,B 0,C 180,E1 25947.964,E2 25947.964} C_VEL
LIN {X 0,Y 539.705,Z 87.802,A -85,B 0,C 180,E1 25944.635,E2 25944.635} C_VEL
LIN {X 0,Y 540.292,Z 69.253,A -85,B 0,C 180,E1 25942.41,E2 25942.41} C_VEL
LIN {X 0,Y 536.463,Z 55.105,A -85,B 0,C 180,E1 25940.366,E2 25940.366} C_VEL
LIN {X 0,Y 536.418,Z 54.977,A -85,B 0,C 180,E1 25937.016,E2 25937.016} C_VEL
LIN {X 0,Y 536.444,Z 54.976,A -85,B 0,C 180,E1 25933.693,E2 25933.693} C_VEL
LIN {X 0,Y 536.461,Z 54.973,A -85,B 0,C 180,E1 25930.307,E2 25930.307} C_VEL
LIN {X 0,Y 536.413,Z 54.976,A -85,B 0,C 180,E1 25927.067,E2 25927.067} C_VEL
LIN {X 0,Y 536.421,Z 54.978,A -85,B 0,C 180,E1 25923.634,E2 25923.634} C_VEL
LIN {X 0,Y 536.469,Z 54.975,A -85,B 0,C 180,E1 25920.321,E2 25920.321} C_VEL
LIN {X 0,Y 536.419,Z 54.976,A -85,B 0,C 180,E1 25917.009,E2 25917.009} C_VEL
LIN {X 0,Y 536.408,Z 54.977,A -85,B 0,C 180,E1 25913.686,E2 25913.686} C_VEL
LIN {X 0,Y 536.455,Z 54.977,A -85,B 0,C 180,E1 25910.388,E2 25910.388} C_VEL
LIN {X 0,Y 536.423,Z 54.976,A -85,B 0,C 180,E1 25907.075,E2 25907.075} C_VEL
LIN {X 0,Y 536.4,Z 54.976,A -85,B 0,C 180,E1 25903.733,E2 25903.733} C_VEL
LIN {X 0,Y 536.444,Z 54.977,A -85,B 0,C 180,E1 25900.511,E2 25900.511} C_VEL
LIN {X 0,Y 536.415,Z 54.977,A -85,B 0,C 180,E1 25897.304,E2 25897.304} C_VEL
LIN {X 0,Y 536.395,Z 54.978,A -85,B 0,C 180,E1 25893.957,E2 25893.957} C_VEL
LIN {X 0,Y 536.43,Z 54.979,A -85,B 0,C 180,E1 25890.646,E2 25890.646} C_VEL
LIN {X 0,Y 536.42,Z 54.978,A -85,B 0,C 180,E1 25887.406,E2 25887.406} C_VEL
LIN {X 0,Y 536.389,Z 54.979,A -85,B 0,C 180,E1 25884.175,E2 25884.175} C_VEL
LIN {X 0,Y 536.438,Z 54.979,A -85,B 0,C 180,E1 25880.95,E2 25880.95} C_VEL
LIN {X 0,Y 536.393,Z 54.98,A -85,B 0,C 180,E1 25877.852,E2 25877.852} C_VEL
LIN {X 0,Y 536.39,Z 54.98,A -85,B 0,C 180,E1 25874.444,E2 25874.444} C_VEL
LIN {X 0,Y 536.44,Z 54.977,A -85,B 0,C 180,E1 25871.144,E2 25871.144} C_VEL
LIN {X 0,Y 536.407,Z 54.982,A -85,B 0,C 180,E1 25867.957,E2 25867.957} C_VEL
LIN {X 0,Y 536.395,Z 54.981,A -85,B 0,C 180,E1 25864.648,E2 25864.648} C_VEL
LIN {X 0,Y 536.465,Z 55.202,A -85,B 0,C 180,E1 25863.214,E2 25863.214} C_VEL
LIN {X 0,Y 541.474,Z 70.092,A -85,B 0,C 180,E1 25861.63,E2 25861.63} C_VEL
LIN {X 0,Y 541.851,Z 72.446,A -85,B 0,C 180,E1 25861.419,E2 25861.419} C_VEL
LIN {X 0,Y 540.529,Z 116.239,A -85,B 0,C 180,E1 25858.074,E2 25858.074} C_VEL
LIN {X 0,Y 539.623,Z 158.682,A -85,B 0,C 180,E1 25854.97,E2 25854.97} C_VEL
LIN {X 0,Y 540.747,Z 169.088,A -85,B 0,C 180,E1 25854.782,E2 25854.782} C_VEL
LIN {X 0,Y 539.943,Z 365.669,A -85,B 0,C 180,E1 25852.113,E2 25852.113} C_VEL
LIN {X 0,Y 539.63,Z 384.775,A -85,B 0,C 180,E1 25851.656,E2 25851.656} C_VEL
LIN {X 0,Y 539.242,Z 403.076,A -85,B 0,C 180,E1 25851.021,E2 25851.021} C_VEL
LIN {X 0,Y 538.798,Z 421.062,A -85,B 0,C 180,E1 25850.192,E2 25850.192} C_VEL
LIN {X 0,Y 538.329,Z 438.219,A -85,B 0,C 180,E1 25849.193,E2 25849.193} C_VEL
LIN {X 0,Y 537.861,Z 454.484,A -85,B 0,C 180,E1 25848.031,E2 25848.031} C_VEL
LIN {X 0,Y 537.4,Z 470.393,A -85,B 0,C 180,E1 25846.651,E2 25846.651} C_VEL
LIN {X 0,Y 536.998,Z 484.131,A -85,B 0,C 180,E1 25845.221,E2 25845.221} C_VEL
LIN {X 0,Y 536.674,Z 496.504,A -85,B 0,C 180,E1 25843.687,E2 25843.687} C_VEL
LIN {X 0,Y 536.408,Z 506.588,A -85,B 0,C 180,E1 25842.16,E2 25842.16} C_VEL
LIN {X 0,Y 536.187,Z 515.96,A -85,B 0,C 180,E1 25840.422,E2 25840.422} C_VEL
LIN {X 0,Y 536.044,Z 523.961,A -85,B 0,C 180,E1 25838.582,E2 25838.582} C_VEL
LIN {X 0,Y 535.956,Z 530.503,A -85,B 0,C 180,E1 25836.643,E2 25836.643} C_VEL
LIN {X 0,Y 535.928,Z 535.255,A -85,B 0,C 180,E1 25834.709,E2 25834.709} C_VEL
LIN {X 0,Y 535.914,Z 538.336,A -85,B 0,C 180,E1 25832.781,E2 25832.781} C_VEL
LIN {X 0,Y 535.917,Z 539.848,A -85,B 0,C 180,E1 25830.749,E2 25830.749} C_VEL
LIN {X 0,Y 535.913,Z 539.618,A -85,B 0,C 180,E1 25828.718,E2 25828.718} C_VEL
LIN {X 0,Y 535.914,Z 537.8,A -85,B 0,C 180,E1 25826.792,E2 25826.792} C_VEL
LIN {X 0,Y 535.933,Z 534.368,A -85,B 0,C 180,E1 25824.863,E2 25824.863} C_VEL
LIN {X 0,Y 535.974,Z 529.233,A -85,B 0,C 180,E1 25822.929,E2 25822.929} C_VEL
LIN {X 0,Y 536.072,Z 522.262,A -85,B 0,C 180,E1 25820.987,E2 25820.987} C_VEL
LIN {X 0,Y 536.235,Z 513.814,A -85,B 0,C 180,E1 25819.146,E2 25819.146} C_VEL
LIN {X 0,Y 536.483,Z 503.952,A -85,B 0,C 180,E1 25817.406,E2 25817.406} C_VEL
LIN {X 0,Y 536.762,Z 493.267,A -85,B 0,C 180,E1 25815.877,E2 25815.877} C_VEL
LIN {X 0,Y 537.14,Z 479.755,A -85,B 0,C 180,E1 25814.287,E2 25814.287} C_VEL
LIN {X 0,Y 537.566,Z 465.174,A -85,B 0,C 180,E1 25812.855,E2 25812.855} C_VEL
LIN {X 0,Y 538.026,Z 449.637,A -85,B 0,C 180,E1 25811.585,E2 25811.585} C_VEL
LIN {X 0,Y 538.509,Z 433.219,A -85,B 0,C 180,E1 25810.477,E2 25810.477} C_VEL
LIN {X 0,Y 538.979,Z 415.775,A -85,B 0,C 180,E1 25809.525,E2 25809.525} C_VEL
LIN {X 0,Y 539.411,Z 397.713,A -85,B 0,C 180,E1 25808.755,E2 25808.755} C_VEL
LIN {X 0,Y 539.79,Z 378.344,A -85,B 0,C 180,E1 25808.15,E2 25808.15} C_VEL
LIN {X 0,Y 540.055,Z 358.924,A -85,B 0,C 180,E1 25807.757,E2 25807.757} C_VEL
LIN {X 0,Y 540.747,Z 160.116,A -85,B 0,C 180,E1 25805.056,E2 25805.056} C_VEL
LIN {X 0,Y 540.426,Z 154.452,A -85,B 0,C 180,E1 25804.934,E2 25804.934} C_VEL
LIN {X 0,Y 541.617,Z 83.124,A -85,B 0,C 180,E1 25801.829,E2 25801.829} C_VEL
LIN {X 0,Y 541.777,Z 69.366,A -85,B 0,C 180,E1 25801.206,E2 25801.206} C_VEL
LIN {X 0,Y 536.562,Z 55.601,A -85,B 0,C 180,E1 25800.27,E2 25800.27} C_VEL
LIN {X 0,Y 536.456,Z 54.992,A -85,B 0,C 180,E1 25800.075,E2 25800.075} C_VEL
LIN {X 0,Y 536.461,Z 54.966,A -85,B 0,C 180,E1 25796.614,E2 25796.614} C_VEL
LIN {X 0,Y 536.449,Z 54.976,A -85,B 0,C 180,E1 25793.254,E2 25793.254} C_VEL
LIN {X 0,Y 536.461,Z 54.976,A -85,B 0,C 180,E1 25789.832,E2 25789.832} C_VEL
LIN {X 0,Y 536.457,Z 54.973,A -85,B 0,C 180,E1 25786.403,E2 25786.403} C_VEL
LIN {X 0,Y 536.454,Z 54.97,A -85,B 0,C 180,E1 25783.013,E2 25783.013} C_VEL
LIN {X 0,Y 536.446,Z 54.974,A -85,B 0,C 180,E1 25779.601,E2 25779.601} C_VEL
LIN {X 0,Y 536.461,Z 54.977,A -85,B 0,C 180,E1 25776.196,E2 25776.196} C_VEL
LIN {X 0,Y 536.462,Z 54.971,A -85,B 0,C 180,E1 25772.718,E2 25772.718} C_VEL
LIN {X 0,Y 536.45,Z 54.97,A -85,B 0,C 180,E1 25769.279,E2 25769.279} C_VEL
LIN {X 0,Y 536.44,Z 54.974,A -85,B 0,C 180,E1 25765.813,E2 25765.813} C_VEL
LIN {X 0,Y 536.465,Z 54.974,A -85,B 0,C 180,E1 25762.42,E2 25762.42} C_VEL
LIN {X 0,Y 536.462,Z 54.969,A -85,B 0,C 180,E1 25758.923,E2 25758.923} C_VEL
LIN {X 0,Y 536.447,Z 54.97,A -85,B 0,C 180,E1 25755.511,E2 25755.511} C_VEL
LIN {X 0,Y 536.434,Z 54.974,A -85,B 0,C 180,E1 25752.049,E2 25752.049} C_VEL
LIN {X 0,Y 536.459,Z 54.974,A -85,B 0,C 180,E1 25748.683,E2 25748.683} C_VEL
LIN {X 0,Y 536.465,Z 54.97,A -85,B 0,C 180,E1 25745.24,E2 25745.24} C_VEL
LIN {X 0,Y 536.44,Z 54.971,A -85,B 0,C 180,E1 25741.816,E2 25741.816} C_VEL
LIN {X 0,Y 536.43,Z 54.974,A -85,B 0,C 180,E1 25738.398,E2 25738.398} C_VEL
LIN {X 0,Y 536.462,Z 54.973,A -85,B 0,C 180,E1 25735.081,E2 25735.081} C_VEL
LIN {X 0,Y 536.464,Z 54.971,A -85,B 0,C 180,E1 25731.641,E2 25731.641} C_VEL
LIN {X 0,Y 536.426,Z 54.973,A -85,B 0,C 180,E1 25728.277,E2 25728.277} C_VEL
LIN {X 0,Y 536.432,Z 54.976,A -85,B 0,C 180,E1 25724.873,E2 25724.873} C_VEL
LIN {X 0,Y 536.467,Z 54.972,A -85,B 0,C 180,E1 25721.528,E2 25721.528} C_VEL
LIN {X 0,Y 536.438,Z 54.97,A -85,B 0,C 180,E1 25718.154,E2 25718.154} C_VEL
LIN {X 0,Y 536.419,Z 54.973,A -85,B 0,C 180,E1 25714.85,E2 25714.85} C_VEL
LIN {X 0,Y 536.454,Z 54.973,A -85,B 0,C 180,E1 25711.501,E2 25711.501} C_VEL
LIN {X 0,Y 536.451,Z 54.97,A -85,B 0,C 180,E1 25708.165,E2 25708.165} C_VEL
LIN {X 0,Y 536.432,Z 54.972,A -85,B 0,C 180,E1 25705.395,E2 25705.395} C_VEL
LIN {X 0,Y 535.426,Z 55.095,A -85,B 0,C 180,E1 25704.573,E2 25704.573} C_VEL
LIN {X 0,Y 528.979,Z 55.914,A -85,B 0,C 180,E1 25702.202,E2 25702.202} C_VEL
LIN {X 0,Y 528.509,Z 55.967,A -85,B 0,C 180,E1 25701.66,E2 25701.66} C_VEL
LIN {X 0,Y 528.518,Z 55.962,A -85,B 0,C 180,E1 25698.247,E2 25698.247} C_VEL
LIN {X 0,Y 528.473,Z 55.965,A -85,B 0,C 180,E1 25694.885,E2 25694.885} C_VEL
LIN {X 0,Y 528.473,Z 55.968,A -85,B 0,C 180,E1 25691.465,E2 25691.465} C_VEL
LIN {X 0,Y 528.527,Z 55.963,A -85,B 0,C 180,E1 25688.213,E2 25688.213} C_VEL
LIN {X 0,Y 528.486,Z 55.97,A -85,B 0,C 180,E1 25684.804,E2 25684.804} C_VEL
LIN {X 0,Y 528.549,Z 56.151,A -85,B 0,C 180,E1 25684.28,E2 25684.28} C_VEL
LIN {X 0,Y 530.478,Z 65.648,A -85,B 0,C 180,E1 25683.189,E2 25683.189} C_VEL
LIN {X 0,Y 530.524,Z 95.895,A -85,B 0,C 180,E1 25680.023,E2 25680.023} C_VEL
LIN {X 0,Y 530.303,Z 127.348,A -85,B 0,C 180,E1 25676.657,E2 25676.657} C_VEL
LIN {X 0,Y 530.004,Z 158.305,A -85,B 0,C 180,E1 25673.337,E2 25673.337} C_VEL
LIN {X 0,Y 529.829,Z 180.565,A -85,B 0,C 180,E1 25670.984,E2 25670.984} C_VEL
LIN {X 0,Y 530.363,Z 186.408,A -85,B 0,C 180,E1 25670.878,E2 25670.878} C_VEL
LIN {X 0,Y 529.916,Z 292.22,A -85,B 0,C 180,E1 25669.408,E2 25669.408} C_VEL
LIN {X 0,Y 529.846,Z 306.448,A -85,B 0,C 180,E1 25669.015,E2 25669.015} C_VEL
LIN {X 0,Y 529.685,Z 320.42,A -85,B 0,C 180,E1 25668.431,E2 25668.431} C_VEL
LIN {X 0,Y 529.421,Z 333.938,A -85,B 0,C 180,E1 25667.644,E2 25667.644} C_VEL
LIN {X 0,Y 529.146,Z 346.291,A -85,B 0,C 180,E1 25666.69,E2 25666.69} C_VEL
LIN {X 0,Y 528.896,Z 357.09,A -85,B 0,C 180,E1 25665.625,E2 25665.625} C_VEL
LIN {X 0,Y 528.637,Z 367.272,A -85,B 0,C 180,E1 25664.345,E2 25664.345} C_VEL
LIN {X 0,Y 528.426,Z 376.092,A -85,B 0,C 180,E1 25662.9,E2 25662.9} C_VEL
LIN {X 0,Y 528.279,Z 383.141,A -85,B 0,C 180,E1 25661.351,E2 25661.351} C_VEL
LIN {X 0,Y 528.194,Z 388.116,A -85,B 0,C 180,E1 25659.808,E2 25659.808} C_VEL
LIN {X 0,Y 528.146,Z 391.328,A -85,B 0,C 180,E1 25658.271,E2 25658.271} C_VEL
LIN {X 0,Y 528.124,Z 393.005,A -85,B 0,C 180,E1 25656.522,E2 25656.522} C_VEL
LIN {X 0,Y 528.126,Z 392.647,A -85,B 0,C 180,E1 25654.777,E2 25654.777} C_VEL
LIN {X 0,Y 528.156,Z 390.258,A -85,B 0,C 180,E1 25653.038,E2 25653.038} C_VEL
LIN {X 0,Y 528.222,Z 386.079,A -85,B 0,C 180,E1 25651.409,E2 25651.409} C_VEL
LIN {X 0,Y 528.326,Z 380.311,A -85,B 0,C 180,E1 25649.891,E2 25649.891} C_VEL
LIN {X 0,Y 528.486,Z 373.092,A -85,B 0,C 180,E1 25648.481,E2 25648.481} C_VEL
LIN {X 0,Y 528.721,Z 363.596,A -85,B 0,C 180,E1 25647.072,E2 25647.072} C_VEL
LIN {X 0,Y 528.995,Z 352.676,A -85,B 0,C 180,E1 25645.826,E2 25645.826} C_VEL
LIN {X 0,Y 529.237,Z 341.104,A -85,B 0,C 180,E1 25644.796,E2 25644.796} C_VEL
LIN {X 0,Y 529.526,Z 328.532,A -85,B 0,C 180,E1 25643.929,E2 25643.929} C_VEL
LIN {X 0,Y 529.737,Z 314.885,A -85,B 0,C 180,E1 25643.225,E2 25643.225} C_VEL
LIN {X 0,Y 529.84,Z 299.717,A -85,B 0,C 180,E1 25642.685,E2 25642.685} C_VEL
LIN {X 0,Y 529.881,Z 284.422,A -85,B 0,C 180,E1 25642.367,E2 25642.367} C_VEL
LIN {X 0,Y 530.22,Z 176.947,A -85,B 0,C 180,E1 25640.885,E2 25640.885} C_VEL
LIN {X 0,Y 530.726,Z 124.571,A -85,B 0,C 180,E1 25637.542,E2 25637.542} C_VEL
LIN {X 0,Y 531.169,Z 72.59,A -85,B 0,C 180,E1 25634.216,E2 25634.216} C_VEL
LIN {X 0,Y 531.084,Z 65.758,A -85,B 0,C 180,E1 25633.775,E2 25633.775} C_VEL
LIN {X 0,Y 529.858,Z 60.866,A -85,B 0,C 180,E1 25633.388,E2 25633.388} C_VEL
LIN {X 0,Y 529.928,Z 60.521,A -85,B 0,C 180,E1 25633.207,E2 25633.207} C_VEL
LIN {X 0,Y 532.406,Z 68.611,A -85,B 0,C 180,E1 25632.457,E2 25632.457} C_VEL
LIN {X 0,Y 531.652,Z 105.682,A -85,B 0,C 180,E1 25629.869,E2 25629.869} C_VEL
LIN {X 0,Y 530.508,Z 158.921,A -85,B 0,C 180,E1 25626.213,E2 25626.213} C_VEL
LIN {X 0,Y 530.325,Z 172.434,A -85,B 0,C 180,E1 25625.32,E2 25625.32} C_VEL
LIN {X 0,Y 530.995,Z 181.664,A -85,B 0,C 180,E1 25625.158,E2 25625.158} C_VEL
LIN {X 0,Y 530.291,Z 289.841,A -85,B 0,C 180,E1 25623.597,E2 25623.597} C_VEL
LIN {X 0,Y 530.136,Z 304.947,A -85,B 0,C 180,E1 25623.175,E2 25623.175} C_VEL
LIN {X 0,Y 529.863,Z 320.066,A -85,B 0,C 180,E1 25622.524,E2 25622.524} C_VEL
LIN {X 0,Y 529.53,Z 333.675,A -85,B 0,C 180,E1 25621.709,E2 25621.709} C_VEL
LIN {X 0,Y 529.233,Z 345.52,A -85,B 0,C 180,E1 25620.791,E2 25620.791} C_VEL
LIN {X 0,Y 528.922,Z 357.025,A -85,B 0,C 180,E1 25619.648,E2 25619.648} C_VEL
LIN {X 0,Y 528.646,Z 366.84,A -85,B 0,C 180,E1 25618.405,E2 25618.405} C_VEL
LIN {X 0,Y 528.451,Z 374.939,A -85,B 0,C 180,E1 25617.11,E2 25617.11} C_VEL
LIN {X 0,Y 528.292,Z 382.067,A -85,B 0,C 180,E1 25615.608,E2 25615.608} C_VEL
LIN {X 0,Y 528.204,Z 387.252,A -85,B 0,C 180,E1 25614.114,E2 25614.114} C_VEL
LIN {X 0,Y 528.15,Z 391.07,A -85,B 0,C 180,E1 25612.44,E2 25612.44} C_VEL
LIN {X 0,Y 528.13,Z 392.921,A -85,B 0,C 180,E1 25610.744,E2 25610.744} C_VEL
LIN {X 0,Y 528.134,Z 392.993,A -85,B 0,C 180,E1 25609.22,E2 25609.22} C_VEL
LIN {X 0,Y 528.166,Z 391.203,A -85,B 0,C 180,E1 25607.481,E2 25607.481} C_VEL
LIN {X 0,Y 528.23,Z 387.572,A -85,B 0,C 180,E1 25605.84,E2 25605.84} C_VEL
LIN {X 0,Y 528.334,Z 382.308,A -85,B 0,C 180,E1 25604.293,E2 25604.293} C_VEL
LIN {X 0,Y 528.506,Z 375.19,A -85,B 0,C 180,E1 25602.78,E2 25602.78} C_VEL
LIN {X 0,Y 528.765,Z 365.857,A -85,B 0,C 180,E1 25601.295,E2 25601.295} C_VEL
LIN {X 0,Y 529.079,Z 355.055,A -85,B 0,C 180,E1 25599.982,E2 25599.982} C_VEL
LIN {X 0,Y 529.399,Z 343.786,A -85,B 0,C 180,E1 25598.91,E2 25598.91} C_VEL
LIN {X 0,Y 529.747,Z 331.233,A -85,B 0,C 180,E1 25597.974,E2 25597.974} C_VEL
LIN {X 0,Y 530.076,Z 316.826,A -85,B 0,C 180,E1 25597.167,E2 25597.167} C_VEL
LIN {X 0,Y 530.32,Z 302.045,A -85,B 0,C 180,E1 25596.582,E2 25596.582} C_VEL
LIN {X 0,Y 530.477,Z 287.195,A -85,B 0,C 180,E1 25596.206,E2 25596.206} C_VEL
LIN {X 0,Y 531.081,Z 182.909,A -85,B 0,C 180,E1 25594.663,E2 25594.663} C_VEL
LIN {X 0,Y 529.703,Z 174.966,A -85,B 0,C 180,E1 25594.458,E2 25594.458} C_VEL
LIN {X 0,Y 530.382,Z 146.014,A -85,B 0,C 180,E1 25591.101,E2 25591.101} C_VEL
LIN {X 0,Y 531.267,Z 116.66,A -85,B 0,C 180,E1 25587.646,E2 25587.646} C_VEL
LIN {X 0,Y 532.272,Z 87.64,A -85,B 0,C 180,E1 25584.174,E2 25584.174} C_VEL
LIN {X 0,Y 532.683,Z 71.187,A -85,B 0,C 180,E1 25582.166,E2 25582.166} C_VEL
LIN {X 0,Y 528.545,Z 56.079,A -85,B 0,C 180,E1 25579.932,E2 25579.932} C_VEL
LIN {X 0,Y 528.502,Z 55.963,A -85,B 0,C 180,E1 25576.486,E2 25576.486} C_VEL
LIN {X 0,Y 528.477,Z 55.966,A -85,B 0,C 180,E1 25573.123,E2 25573.123} C_VEL
LIN {X 0,Y 528.505,Z 55.965,A -85,B 0,C 180,E1 25569.804,E2 25569.804} C_VEL
LIN {X 0,Y 528.522,Z 55.963,A -85,B 0,C 180,E1 25566.409,E2 25566.409} C_VEL
LIN {X 0,Y 528.477,Z 55.965,A -85,B 0,C 180,E1 25563.037,E2 25563.037} C_VEL
LIN {X 0,Y 528.473,Z 55.966,A -85,B 0,C 180,E1 25559.567,E2 25559.567} C_VEL
LIN {X 0,Y 528.519,Z 55.966,A -85,B 0,C 180,E1 25556.312,E2 25556.312} C_VEL
LIN {X 0,Y 528.482,Z 55.965,A -85,B 0,C 180,E1 25553.046,E2 25553.046} C_VEL
LIN {X 0,Y 528.465,Z 55.966,A -85,B 0,C 180,E1 25549.646,E2 25549.646} C_VEL
LIN {X 0,Y 528.498,Z 55.966,A -85,B 0,C 180,E1 25546.321,E2 25546.321} C_VEL
LIN {X 0,Y 528.491,Z 55.964,A -85,B 0,C 180,E1 25543.061,E2 25543.061} C_VEL
LIN {X 0,Y 528.46,Z 55.965,A -85,B 0,C 180,E1 25539.743,E2 25539.743} C_VEL
LIN {X 0,Y 528.488,Z 55.968,A -85,B 0,C 180,E1 25536.472,E2 25536.472} C_VEL
LIN {X 0,Y 528.501,Z 55.967,A -85,B 0,C 180,E1 25533.118,E2 25533.118} C_VEL
LIN {X 0,Y 528.454,Z 55.967,A -85,B 0,C 180,E1 25529.844,E2 25529.844} C_VEL
LIN {X 0,Y 528.465,Z 55.968,A -85,B 0,C 180,E1 25526.464,E2 25526.464} C_VEL
LIN {X 0,Y 528.511,Z 55.967,A -85,B 0,C 180,E1 25523.151,E2 25523.151} C_VEL
LIN {X 0,Y 528.456,Z 55.969,A -85,B 0,C 180,E1 25519.821,E2 25519.821} C_VEL
LIN {X 0,Y 528.45,Z 55.967,A -85,B 0,C 180,E1 25516.441,E2 25516.441} C_VEL
LIN {X 0,Y 528.51,Z 55.964,A -85,B 0,C 180,E1 25513.224,E2 25513.224} C_VEL
LIN {X 0,Y 528.464,Z 55.97,A -85,B 0,C 180,E1 25509.981,E2 25509.981} C_VEL
LIN {X 0,Y 528.455,Z 55.971,A -85,B 0,C 180,E1 25506.584,E2 25506.584} C_VEL
LIN {X 0,Y 528.542,Z 56.215,A -85,B 0,C 180,E1 25503.658,E2 25503.658} C_VEL
LIN {X 0,Y 534.561,Z 74.312,A -85,B 0,C 180,E1 25501.708,E2 25501.708} C_VEL
LIN {X 0,Y 533.093,Z 116.155,A -85,B 0,C 180,E1 25498.451,E2 25498.451} C_VEL
LIN {X 0,Y 531.979,Z 158.616,A -85,B 0,C 180,E1 25495.27,E2 25495.27} C_VEL
LIN {X 0,Y 533.207,Z 169.991,A -85,B 0,C 180,E1 25495.058,E2 25495.058} C_VEL
LIN {X 0,Y 532.305,Z 365.032,A -85,B 0,C 180,E1 25492.379,E2 25492.379} C_VEL
LIN {X 0,Y 531.95,Z 384.067,A -85,B 0,C 180,E1 25491.918,E2 25491.918} C_VEL
LIN {X 0,Y 531.524,Z 402.054,A -85,B 0,C 180,E1 25491.288,E2 25491.288} C_VEL
LIN {X 0,Y 531.062,Z 419.144,A -85,B 0,C 180,E1 25490.5,E2 25490.5} C_VEL
LIN {X 0,Y 530.537,Z 436.504,A -85,B 0,C 180,E1 25489.487,E2 25489.487} C_VEL
LIN {X 0,Y 530.039,Z 452.217,A -85,B 0,C 180,E1 25488.363,E2 25488.363} C_VEL
LIN {X 0,Y 529.546,Z 467.769,A -85,B 0,C 180,E1 25487.018,E2 25487.018} C_VEL
LIN {X 0,Y 529.101,Z 481.777,A -85,B 0,C 180,E1 25485.566,E2 25485.566} C_VEL
LIN {X 0,Y 528.736,Z 494.382,A -85,B 0,C 180,E1 25484.008,E2 25484.008} C_VEL
LIN {X 0,Y 528.438,Z 505.622,A -85,B 0,C 180,E1 25482.346,E2 25482.346} C_VEL
LIN {X 0,Y 528.209,Z 515.483,A -85,B 0,C 180,E1 25480.581,E2 25480.581} C_VEL
LIN {X 0,Y 528.059,Z 523.762,A -85,B 0,C 180,E1 25478.741,E2 25478.741} C_VEL
LIN {X 0,Y 527.979,Z 529.897,A -85,B 0,C 180,E1 25476.962,E2 25476.962} C_VEL
LIN {X 0,Y 527.933,Z 534.841,A -85,B 0,C 180,E1 25474.999,E2 25474.999} C_VEL
LIN {X 0,Y 527.915,Z 538.221,A -85,B 0,C 180,E1 25472.932,E2 25472.932} C_VEL
LIN {X 0,Y 527.916,Z 539.825,A -85,B 0,C 180,E1 25470.869,E2 25470.869} C_VEL
LIN {X 0,Y 527.913,Z 539.686,A -85,B 0,C 180,E1 25468.807,E2 25468.807} C_VEL
LIN {X 0,Y 527.916,Z 537.959,A -85,B 0,C 180,E1 25466.852,E2 25466.852} C_VEL
LIN {X 0,Y 527.935,Z 534.368,A -85,B 0,C 180,E1 25464.785,E2 25464.785} C_VEL
LIN {X 0,Y 527.982,Z 529.232,A -85,B 0,C 180,E1 25462.821,E2 25462.821} C_VEL
LIN {X 0,Y 528.083,Z 522.579,A -85,B 0,C 180,E1 25460.959,E2 25460.959} C_VEL
LIN {X 0,Y 528.244,Z 513.837,A -85,B 0,C 180,E1 25459.09,E2 25459.09} C_VEL
LIN {X 0,Y 528.495,Z 503.629,A -85,B 0,C 180,E1 25457.324,E2 25457.324} C_VEL
LIN {X 0,Y 528.807,Z 492.007,A -85,B 0,C 180,E1 25455.66,E2 25455.66} C_VEL
LIN {X 0,Y 529.203,Z 478.846,A -85,B 0,C 180,E1 25454.089,E2 25454.089} C_VEL
LIN {X 0,Y 529.665,Z 464.411,A -85,B 0,C 180,E1 25452.648,E2 25452.648} C_VEL
LIN {X 0,Y 530.175,Z 448.901,A -85,B 0,C 180,E1 25451.359,E2 25451.359} C_VEL
LIN {X 0,Y 530.712,Z 432.507,A -85,B 0,C 180,E1 25450.235,E2 25450.235} C_VEL
LIN {X 0,Y 531.234,Z 415.253,A -85,B 0,C 180,E1 25449.279,E2 25449.279} C_VEL
LIN {X 0,Y 531.728,Z 397.027,A -85,B 0,C 180,E1 25448.49,E2 25448.49} C_VEL
LIN {X 0,Y 532.153,Z 377.783,A -85,B 0,C 180,E1 25447.882,E2 25447.882} C_VEL
LIN {X 0,Y 532.445,Z 358.401,A -85,B 0,C 180,E1 25447.485,E2 25447.485} C_VEL
LIN {X 0,Y 533.247,Z 160.812,A -85,B 0,C 180,E1 25444.766,E2 25444.766} C_VEL
LIN {X 0,Y 532.889,Z 154.983,A -85,B 0,C 180,E1 25444.651,E2 25444.651} C_VEL
LIN {X 0,Y 534.44,Z 77.464,A -85,B 0,C 180,E1 25441.202,E2 25441.202} C_VEL
LIN {X 0,Y 534.307,Z 71.473,A -85,B 0,C 180,E1 25440.916,E2 25440.916} C_VEL
LIN {X 0,Y 528.609,Z 56.537,A -85,B 0,C 180,E1 25439.883,E2 25439.883} C_VEL
LIN {X 0,Y 528.525,Z 55.962,A -85,B 0,C 180,E1 25439.663,E2 25439.663} C_VEL
LIN {X 0,Y 528.515,Z 55.958,A -85,B 0,C 180,E1 25436.151,E2 25436.151} C_VEL
LIN {X 0,Y 528.519,Z 55.961,A -85,B 0,C 180,E1 25432.746,E2 25432.746} C_VEL
LIN {X 0,Y 528.511,Z 55.964,A -85,B 0,C 180,E1 25429.343,E2 25429.343} C_VEL
LIN {X 0,Y 528.524,Z 55.964,A -85,B 0,C 180,E1 25425.881,E2 25425.881} C_VEL
LIN {X 0,Y 528.519,Z 55.961,A -85,B 0,C 180,E1 25422.457,E2 25422.457} C_VEL
LIN {X 0,Y 528.516,Z 55.959,A -85,B 0,C 180,E1 25419.048,E2 25419.048} C_VEL
LIN {X 0,Y 528.504,Z 55.96,A -85,B 0,C 180,E1 25415.563,E2 25415.563} C_VEL
LIN {X 0,Y 528.523,Z 55.963,A -85,B 0,C 180,E1 25412.113,E2 25412.113} C_VEL
LIN {X 0,Y 528.523,Z 55.962,A -85,B 0,C 180,E1 25408.626,E2 25408.626} C_VEL
LIN {X 0,Y 528.518,Z 55.959,A -85,B 0,C 180,E1 25405.192,E2 25405.192} C_VEL
LIN {X 0,Y 528.499,Z 55.962,A -85,B 0,C 180,E1 25401.738,E2 25401.738} C_VEL
LIN {X 0,Y 528.51,Z 55.964,A -85,B 0,C 180,E1 25398.254,E2 25398.254} C_VEL
LIN {X 0,Y 528.525,Z 55.962,A -85,B 0,C 180,E1 25394.797,E2 25394.797} C_VEL
LIN {X 0,Y 528.521,Z 55.959,A -85,B 0,C 180,E1 25391.347,E2 25391.347} C_VEL
LIN {X 0,Y 528.496,Z 55.961,A -85,B 0,C 180,E1 25387.938,E2 25387.938} C_VEL
LIN {X 0,Y 528.501,Z 55.962,A -85,B 0,C 180,E1 25384.449,E2 25384.449} C_VEL
LIN {X 0,Y 528.528,Z 55.964,A -85,B 0,C 180,E1 25380.975,E2 25380.975} C_VEL
LIN {X 0,Y 528.523,Z 55.96,A -85,B 0,C 180,E1 25377.506,E2 25377.506} C_VEL
LIN {X 0,Y 528.49,Z 55.96,A -85,B 0,C 180,E1 25374.136,E2 25374.136} C_VEL
LIN {X 0,Y 528.491,Z 55.961,A -85,B 0,C 180,E1 25370.636,E2 25370.636} C_VEL
LIN {X 0,Y 528.522,Z 55.964,A -85,B 0,C 180,E1 25367.212,E2 25367.212} C_VEL
LIN {X 0,Y 528.523,Z 55.961,A -85,B 0,C 180,E1 25363.74,E2 25363.74} C_VEL
LIN {X 0,Y 528.485,Z 55.962,A -85,B 0,C 180,E1 25360.416,E2 25360.416} C_VEL
LIN {X 0,Y 528.486,Z 55.952,A -85,B 0,C 180,E1 25356.944,E2 25356.944} C_VEL
LIN {X 0,Y 528.525,Z 55.963,A -85,B 0,C 180,E1 25353.604,E2 25353.604} C_VEL
LIN {X 0,Y 528.498,Z 55.957,A -85,B 0,C 180,E1 25350.267,E2 25350.267} C_VEL
LIN {X 0,Y 528.477,Z 55.965,A -85,B 0,C 180,E1 25346.941,E2 25346.941} C_VEL
LIN {X 0,Y 528.502,Z 55.964,A -85,B 0,C 180,E1 25343.555,E2 25343.555} C_VEL
LIN {X 0,Y 528.509,Z 55.967,A -85,B 0,C 180,E1 25341.66,E2 25341.66} C_VEL
LIN {X 0,Y 527.48,Z 56.088,A -85,B 0,C 180,E1 25340.825,E2 25340.825} C_VEL
LIN {X 0,Y 521.026,Z 56.899,A -85,B 0,C 180,E1 25338.419,E2 25338.419} C_VEL
LIN {X 0,Y 520.579,Z 56.956,A -85,B 0,C 180,E1 25337.869,E2 25337.869} C_VEL
LIN {X 0,Y 520.56,Z 56.953,A -85,B 0,C 180,E1 25334.511,E2 25334.511} C_VEL
LIN {X 0,Y 520.528,Z 56.956,A -85,B 0,C 180,E1 25331.151,E2 25331.151} C_VEL
LIN {X 0,Y 520.549,Z 56.958,A -85,B 0,C 180,E1 25327.785,E2 25327.785} C_VEL
LIN {X 0,Y 520.603,Z 57.199,A -85,B 0,C 180,E1 25324.54,E2 25324.54} C_VEL
LIN {X 0,Y 522.833,Z 67.491,A -85,B 0,C 180,E1 25323.352,E2 25323.352} C_VEL
LIN {X 0,Y 522.841,Z 98.047,A -85,B 0,C 180,E1 25320.137,E2 25320.137} C_VEL
LIN {X 0,Y 522.592,Z 129.219,A -85,B 0,C 180,E1 25316.784,E2 25316.784} C_VEL
LIN {X 0,Y 522.263,Z 161.259,A -85,B 0,C 180,E1 25313.345,E2 25313.345} C_VEL
LIN {X 0,Y 522.134,Z 181.559,A -85,B 0,C 180,E1 25311.21,E2 25311.21} C_VEL
LIN {X 0,Y 522.662,Z 187.125,A -85,B 0,C 180,E1 25311.107,E2 25311.107} C_VEL
LIN {X 0,Y 522.174,Z 293.194,A -85,B 0,C 180,E1 25309.612,E2 25309.612} C_VEL
LIN {X 0,Y 522.113,Z 307,A -85,B 0,C 180,E1 25309.23,E2 25309.23} C_VEL
LIN {X 0,Y 521.952,Z 320.761,A -85,B 0,C 180,E1 25308.656,E2 25308.656} C_VEL
LIN {X 0,Y 521.669,Z 334.458,A -85,B 0,C 180,E1 25307.857,E2 25307.857} C_VEL
LIN {X 0,Y 521.385,Z 346.315,A -85,B 0,C 180,E1 25306.946,E2 25306.946} C_VEL
LIN {X 0,Y 521.113,Z 357.353,A -85,B 0,C 180,E1 25305.866,E2 25305.866} C_VEL
LIN {X 0,Y 520.816,Z 367.714,A -85,B 0,C 180,E1 25304.565,E2 25304.565} C_VEL
LIN {X 0,Y 520.575,Z 376.422,A -85,B 0,C 180,E1 25303.146,E2 25303.146} C_VEL
LIN {X 0,Y 520.415,Z 382.988,A -85,B 0,C 180,E1 25301.75,E2 25301.75} C_VEL
LIN {X 0,Y 520.308,Z 388.382,A -85,B 0,C 180,E1 25300.182,E2 25300.182} C_VEL
LIN {X 0,Y 520.233,Z 392.098,A -85,B 0,C 180,E1 25298.509,E2 25298.509} C_VEL
LIN {X 0,Y 520.201,Z 393.931,A -85,B 0,C 180,E1 25296.843,E2 25296.843} C_VEL
LIN {X 0,Y 520.197,Z 393.991,A -85,B 0,C 180,E1 25295.182,E2 25295.182} C_VEL
LIN {X 0,Y 520.224,Z 392.289,A -85,B 0,C 180,E1 25293.525,E2 25293.525} C_VEL
LIN {X 0,Y 520.298,Z 388.435,A -85,B 0,C 180,E1 25291.761,E2 25291.761} C_VEL
LIN {X 0,Y 520.412,Z 382.731,A -85,B 0,C 180,E1 25290.109,E2 25290.109} C_VEL
LIN {X 0,Y 520.578,Z 375.893,A -85,B 0,C 180,E1 25288.679,E2 25288.679} C_VEL
LIN {X 0,Y 520.803,Z 367.732,A -85,B 0,C 180,E1 25287.358,E2 25287.358} C_VEL
LIN {X 0,Y 521.099,Z 357.204,A -85,B 0,C 180,E1 25286.038,E2 25286.038} C_VEL
LIN {X 0,Y 521.391,Z 345.29,A -85,B 0,C 180,E1 25284.883,E2 25284.883} C_VEL
LIN {X 0,Y 521.691,Z 332.757,A -85,B 0,C 180,E1 25283.948,E2 25283.948} C_VEL
LIN {X 0,Y 521.944,Z 320.211,A -85,B 0,C 180,E1 25283.233,E2 25283.233} C_VEL
LIN {X 0,Y 522.082,Z 305.101,A -85,B 0,C 180,E1 25282.617,E2 25282.617} C_VEL
LIN {X 0,Y 522.133,Z 289.331,A -85,B 0,C 180,E1 25282.223,E2 25282.223} C_VEL
LIN {X 0,Y 522.548,Z 177.781,A -85,B 0,C 180,E1 25280.653,E2 25280.653} C_VEL
LIN {X 0,Y 523.069,Z 124.373,A -85,B 0,C 180,E1 25277.244,E2 25277.244} C_VEL
LIN {X 0,Y 523.531,Z 72.645,A -85,B 0,C 180,E1 25273.923,E2 25273.923} C_VEL
LIN {X 0,Y 523.31,Z 67.206,A -85,B 0,C 180,E1 25273.567,E2 25273.567} C_VEL
LIN {X 0,Y 522.916,Z 65.2,A -85,B 0,C 180,E1 25273.347,E2 25273.347} C_VEL
LIN {X 0,Y 523.176,Z 65.282,A -85,B 0,C 180,E1 25273.198,E2 25273.198} C_VEL
LIN {X 0,Y 525.095,Z 71.756,A -85,B 0,C 180,E1 25272.605,E2 25272.605} C_VEL
LIN {X 0,Y 523.721,Z 123.076,A -85,B 0,C 180,E1 25269,E2 25269} C_VEL
LIN {X 0,Y 522.664,Z 172.257,A -85,B 0,C 180,E1 25265.619,E2 25265.619} C_VEL
LIN {X 0,Y 523.443,Z 182.112,A -85,B 0,C 180,E1 25265.441,E2 25265.441} C_VEL
LIN {X 0,Y 522.64,Z 290.533,A -85,B 0,C 180,E1 25263.842,E2 25263.842} C_VEL
LIN {X 0,Y 522.479,Z 304.911,A -85,B 0,C 180,E1 25263.438,E2 25263.438} C_VEL
LIN {X 0,Y 522.192,Z 319.605,A -85,B 0,C 180,E1 25262.808,E2 25262.808} C_VEL
LIN {X 0,Y 521.856,Z 332.733,A -85,B 0,C 180,E1 25262.039,E2 25262.039} C_VEL
LIN {X 0,Y 521.493,Z 345.686,A -85,B 0,C 180,E1 25261.045,E2 25261.045} C_VEL
LIN {X 0,Y 521.148,Z 357.073,A -85,B 0,C 180,E1 25259.915,E2 25259.915} C_VEL
LIN {X 0,Y 520.844,Z 366.943,A -85,B 0,C 180,E1 25258.679,E2 25258.679} C_VEL
LIN {X 0,Y 520.584,Z 376.104,A -85,B 0,C 180,E1 25257.205,E2 25257.205} C_VEL
LIN {X 0,Y 520.398,Z 383.52,A -85,B 0,C 180,E1 25255.606,E2 25255.606} C_VEL
LIN {X 0,Y 520.287,Z 388.808,A -85,B 0,C 180,E1 25254.004,E2 25254.004} C_VEL
LIN {X 0,Y 520.232,Z 392.188,A -85,B 0,C 180,E1 25252.464,E2 25252.464} C_VEL
LIN {X 0,Y 520.207,Z 394.02,A -85,B 0,C 180,E1 25250.768,E2 25250.768} C_VEL
LIN {X 0,Y 520.213,Z 394.101,A -85,B 0,C 180,E1 25249.195,E2 25249.195} C_VEL
LIN {X 0,Y 520.254,Z 392.311,A -85,B 0,C 180,E1 25247.429,E2 25247.429} C_VEL
LIN {X 0,Y 520.332,Z 388.701,A -85,B 0,C 180,E1 25245.77,E2 25245.77} C_VEL
LIN {X 0,Y 520.457,Z 383.516,A -85,B 0,C 180,E1 25244.217,E2 25244.217} C_VEL
LIN {X 0,Y 520.657,Z 376.436,A -85,B 0,C 180,E1 25242.68,E2 25242.68} C_VEL
LIN {X 0,Y 520.95,Z 367.143,A -85,B 0,C 180,E1 25241.172,E2 25241.172} C_VEL
LIN {X 0,Y 521.285,Z 356.907,A -85,B 0,C 180,E1 25239.895,E2 25239.895} C_VEL
LIN {X 0,Y 521.638,Z 345.986,A -85,B 0,C 180,E1 25238.814,E2 25238.814} C_VEL
LIN {X 0,Y 522.042,Z 332.819,A -85,B 0,C 180,E1 25237.799,E2 25237.799} C_VEL
LIN {X 0,Y 522.381,Z 319.264,A -85,B 0,C 180,E1 25237.011,E2 25237.011} C_VEL
LIN {X 0,Y 522.663,Z 304.914,A -85,B 0,C 180,E1 25236.403,E2 25236.403} C_VEL
LIN {X 0,Y 522.859,Z 289.232,A -85,B 0,C 180,E1 25235.971,E2 25235.971} C_VEL
LIN {X 0,Y 523.598,Z 184.053,A -85,B 0,C 180,E1 25234.37,E2 25234.37} C_VEL
LIN {X 0,Y 521.989,Z 174.858,A -85,B 0,C 180,E1 25234.13,E2 25234.13} C_VEL
LIN {X 0,Y 522.769,Z 145.729,A -85,B 0,C 180,E1 25230.709,E2 25230.709} C_VEL
LIN {X 0,Y 523.731,Z 116.924,A -85,B 0,C 180,E1 25227.27,E2 25227.27} C_VEL
LIN {X 0,Y 524.833,Z 87.987,A -85,B 0,C 180,E1 25223.762,E2 25223.762} C_VEL
LIN {X 0,Y 525.263,Z 73.928,A -85,B 0,C 180,E1 25222.024,E2 25222.024} C_VEL
LIN {X 0,Y 520.58,Z 57.08,A -85,B 0,C 180,E1 25219.492,E2 25219.492} C_VEL
LIN {X 0,Y 520.59,Z 56.952,A -85,B 0,C 180,E1 25216.056,E2 25216.056} C_VEL
LIN {X 0,Y 520.554,Z 56.953,A -85,B 0,C 180,E1 25212.645,E2 25212.645} C_VEL
LIN {X 0,Y 520.536,Z 56.952,A -85,B 0,C 180,E1 25209.285,E2 25209.285} C_VEL
LIN {X 0,Y 520.572,Z 56.956,A -85,B 0,C 180,E1 25205.954,E2 25205.954} C_VEL
LIN {X 0,Y 520.575,Z 56.953,A -85,B 0,C 180,E1 25202.532,E2 25202.532} C_VEL
LIN {X 0,Y 520.532,Z 56.954,A -85,B 0,C 180,E1 25199.23,E2 25199.23} C_VEL
LIN {X 0,Y 520.535,Z 56.955,A -85,B 0,C 180,E1 25195.704,E2 25195.704} C_VEL
LIN {X 0,Y 520.578,Z 56.954,A -85,B 0,C 180,E1 25192.334,E2 25192.334} C_VEL
LIN {X 0,Y 520.557,Z 56.954,A -85,B 0,C 180,E1 25188.926,E2 25188.926} C_VEL
LIN {X 0,Y 520.524,Z 56.954,A -85,B 0,C 180,E1 25185.653,E2 25185.653} C_VEL
LIN {X 0,Y 520.549,Z 56.954,A -85,B 0,C 180,E1 25182.308,E2 25182.308} C_VEL
LIN {X 0,Y 520.571,Z 56.953,A -85,B 0,C 180,E1 25178.951,E2 25178.951} C_VEL
LIN {X 0,Y 520.523,Z 56.956,A -85,B 0,C 180,E1 25175.607,E2 25175.607} C_VEL
LIN {X 0,Y 520.518,Z 56.956,A -85,B 0,C 180,E1 25172.081,E2 25172.081} C_VEL
LIN {X 0,Y 520.56,Z 56.957,A -85,B 0,C 180,E1 25168.762,E2 25168.762} C_VEL
LIN {X 0,Y 520.549,Z 56.956,A -85,B 0,C 180,E1 25165.351,E2 25165.351} C_VEL
LIN {X 0,Y 520.51,Z 56.957,A -85,B 0,C 180,E1 25162.07,E2 25162.07} C_VEL
LIN {X 0,Y 520.527,Z 56.958,A -85,B 0,C 180,E1 25158.682,E2 25158.682} C_VEL
LIN {X 0,Y 520.571,Z 56.953,A -85,B 0,C 180,E1 25155.289,E2 25155.289} C_VEL
LIN {X 0,Y 520.523,Z 56.959,A -85,B 0,C 180,E1 25151.949,E2 25151.949} C_VEL
LIN {X 0,Y 520.516,Z 56.96,A -85,B 0,C 180,E1 25148.574,E2 25148.574} C_VEL
LIN {X 0,Y 520.565,Z 56.957,A -85,B 0,C 180,E1 25145.283,E2 25145.283} C_VEL
LIN {X 0,Y 520.568,Z 57.251,A -85,B 0,C 180,E1 25144.124,E2 25144.124} C_VEL
LIN {X 0,Y 526.681,Z 74.954,A -85,B 0,C 180,E1 25142.146,E2 25142.146} C_VEL
LIN {X 0,Y 527.211,Z 77.768,A -85,B 0,C 180,E1 25141.876,E2 25141.876} C_VEL
LIN {X 0,Y 525.505,Z 120.669,A -85,B 0,C 180,E1 25138.475,E2 25138.475} C_VEL
LIN {X 0,Y 524.419,Z 159.214,A -85,B 0,C 180,E1 25135.562,E2 25135.562} C_VEL
LIN {X 0,Y 525.682,Z 170.851,A -85,B 0,C 180,E1 25135.343,E2 25135.343} C_VEL
LIN {X 0,Y 524.675,Z 364.562,A -85,B 0,C 180,E1 25132.648,E2 25132.648} C_VEL
LIN {X 0,Y 524.282,Z 383.432,A -85,B 0,C 180,E1 25132.186,E2 25132.186} C_VEL
LIN {X 0,Y 523.798,Z 401.814,A -85,B 0,C 180,E1 25131.53,E2 25131.53} C_VEL
LIN {X 0,Y 523.272,Z 419.306,A -85,B 0,C 180,E1 25130.702,E2 25130.702} C_VEL
LIN {X 0,Y 522.697,Z 436.473,A -85,B 0,C 180,E1 25129.675,E2 25129.675} C_VEL
LIN {X 0,Y 522.12,Z 452.872,A -85,B 0,C 180,E1 25128.466,E2 25128.466} C_VEL
LIN {X 0,Y 521.576,Z 468.614,A -85,B 0,C 180,E1 25127.056,E2 25127.056} C_VEL
LIN {X 0,Y 521.108,Z 482.323,A -85,B 0,C 180,E1 25125.583,E2 25125.583} C_VEL
LIN {X 0,Y 520.708,Z 495.477,A -85,B 0,C 180,E1 25123.889,E2 25123.889} C_VEL
LIN {X 0,Y 520.414,Z 506.349,A -85,B 0,C 180,E1 25122.202,E2 25122.202} C_VEL
LIN {X 0,Y 520.2,Z 515.877,A -85,B 0,C 180,E1 25120.41,E2 25120.41} C_VEL
LIN {X 0,Y 520.072,Z 523.992,A -85,B 0,C 180,E1 25118.514,E2 25118.514} C_VEL
LIN {X 0,Y 519.979,Z 530.266,A -85,B 0,C 180,E1 25116.626,E2 25116.626} C_VEL
LIN {X 0,Y 519.938,Z 535.085,A -85,B 0,C 180,E1 25114.633,E2 25114.633} C_VEL
LIN {X 0,Y 519.919,Z 538.267,A -85,B 0,C 180,E1 25112.536,E2 25112.536} C_VEL
LIN {X 0,Y 519.917,Z 539.555,A -85,B 0,C 180,E1 25110.552,E2 25110.552} C_VEL
LIN {X 0,Y 519.919,Z 539.121,A -85,B 0,C 180,E1 25108.458,E2 25108.458} C_VEL
LIN {X 0,Y 519.923,Z 536.838,A -85,B 0,C 180,E1 25106.362,E2 25106.362} C_VEL
LIN {X 0,Y 519.952,Z 532.918,A -85,B 0,C 180,E1 25104.373,E2 25104.373} C_VEL
LIN {X 0,Y 520.024,Z 527.193,A -85,B 0,C 180,E1 25102.377,E2 25102.377} C_VEL
LIN {X 0,Y 520.134,Z 519.514,A -85,B 0,C 180,E1 25100.374,E2 25100.374} C_VEL
LIN {X 0,Y 520.321,Z 510.257,A -85,B 0,C 180,E1 25098.473,E2 25098.473} C_VEL
LIN {X 0,Y 520.611,Z 499.486,A -85,B 0,C 180,E1 25096.677,E2 25096.677} C_VEL
LIN {X 0,Y 520.966,Z 487.225,A -85,B 0,C 180,E1 25094.985,E2 25094.985} C_VEL
LIN {X 0,Y 521.403,Z 474.354,A -85,B 0,C 180,E1 25093.499,E2 25093.499} C_VEL
LIN {X 0,Y 521.913,Z 459.867,A -85,B 0,C 180,E1 25092.094,E2 25092.094} C_VEL
LIN {X 0,Y 522.474,Z 444.367,A -85,B 0,C 180,E1 25090.842,E2 25090.842} C_VEL
LIN {X 0,Y 523.051,Z 428.079,A -85,B 0,C 180,E1 25089.759,E2 25089.759} C_VEL
LIN {X 0,Y 523.604,Z 411.062,A -85,B 0,C 180,E1 25088.845,E2 25088.845} C_VEL
LIN {X 0,Y 524.14,Z 392.742,A -85,B 0,C 180,E1 25088.084,E2 25088.084} C_VEL
LIN {X 0,Y 524.598,Z 373.943,A -85,B 0,C 180,E1 25087.52,E2 25087.52} C_VEL
LIN {X 0,Y 524.885,Z 354.358,A -85,B 0,C 180,E1 25087.15,E2 25087.15} C_VEL
LIN {X 0,Y 525.761,Z 161.485,A -85,B 0,C 180,E1 25084.467,E2 25084.467} C_VEL
LIN {X 0,Y 525.384,Z 154.53,A -85,B 0,C 180,E1 25084.316,E2 25084.316} C_VEL
LIN {X 0,Y 527.15,Z 77.581,A -85,B 0,C 180,E1 25080.828,E2 25080.828} C_VEL
LIN {X 0,Y 527.044,Z 74.142,A -85,B 0,C 180,E1 25080.659,E2 25080.659} C_VEL
LIN {X 0,Y 520.668,Z 57.463,A -85,B 0,C 180,E1 25079.482,E2 25079.482} C_VEL
LIN {X 0,Y 520.577,Z 56.952,A -85,B 0,C 180,E1 25079.278,E2 25079.278} C_VEL
LIN {X 0,Y 520.584,Z 56.951,A -85,B 0,C 180,E1 25075.756,E2 25075.756} C_VEL
LIN {X 0,Y 520.579,Z 56.952,A -85,B 0,C 180,E1 25072.217,E2 25072.217} C_VEL
LIN {X 0,Y 520.582,Z 56.949,A -85,B 0,C 180,E1 25068.795,E2 25068.795} C_VEL
LIN {X 0,Y 520.57,Z 56.952,A -85,B 0,C 180,E1 25065.288,E2 25065.288} C_VEL
LIN {X 0,Y 520.579,Z 56.952,A -85,B 0,C 180,E1 25061.795,E2 25061.795} C_VEL
LIN {X 0,Y 520.582,Z 56.952,A -85,B 0,C 180,E1 25058.343,E2 25058.343} C_VEL
LIN {X 0,Y 520.585,Z 56.945,A -85,B 0,C 180,E1 25054.907,E2 25054.907} C_VEL
LIN {X 0,Y 520.565,Z 56.948,A -85,B 0,C 180,E1 25051.486,E2 25051.486} C_VEL
LIN {X 0,Y 520.57,Z 56.951,A -85,B 0,C 180,E1 25047.947,E2 25047.947} C_VEL
LIN {X 0,Y 520.585,Z 56.953,A -85,B 0,C 180,E1 25044.446,E2 25044.446} C_VEL
LIN {X 0,Y 520.587,Z 56.949,A -85,B 0,C 180,E1 25040.931,E2 25040.931} C_VEL
LIN {X 0,Y 520.565,Z 56.949,A -85,B 0,C 180,E1 25037.551,E2 25037.551} C_VEL
LIN {X 0,Y 520.559,Z 56.95,A -85,B 0,C 180,E1 25034.084,E2 25034.084} C_VEL
LIN {X 0,Y 520.58,Z 56.952,A -85,B 0,C 180,E1 25030.625,E2 25030.625} C_VEL
LIN {X 0,Y 520.588,Z 56.949,A -85,B 0,C 180,E1 25027.171,E2 25027.171} C_VEL
LIN {X 0,Y 520.564,Z 56.946,A -85,B 0,C 180,E1 25023.744,E2 25023.744} C_VEL
LIN {X 0,Y 520.552,Z 56.948,A -85,B 0,C 180,E1 25020.33,E2 25020.33} C_VEL
LIN {X 0,Y 520.577,Z 56.954,A -85,B 0,C 180,E1 25016.917,E2 25016.917} C_VEL
LIN {X 0,Y 520.589,Z 56.948,A -85,B 0,C 180,E1 25013.493,E2 25013.493} C_VEL
LIN {X 0,Y 520.557,Z 56.946,A -85,B 0,C 180,E1 25010.045,E2 25010.045} C_VEL
LIN {X 0,Y 520.546,Z 56.949,A -85,B 0,C 180,E1 25006.56,E2 25006.56} C_VEL
LIN {X 0,Y 520.57,Z 56.952,A -85,B 0,C 180,E1 25003.14,E2 25003.14} C_VEL
LIN {X 0,Y 520.589,Z 56.951,A -85,B 0,C 180,E1 24999.657,E2 24999.657} C_VEL
LIN {X 0,Y 520.55,Z 56.938,A -85,B 0,C 180,E1 24996.331,E2 24996.331} C_VEL
LIN {X 0,Y 520.543,Z 56.954,A -85,B 0,C 180,E1 24992.92,E2 24992.92} C_VEL
LIN {X 0,Y 520.576,Z 56.945,A -85,B 0,C 180,E1 24989.531,E2 24989.531} C_VEL
LIN {X 0,Y 520.583,Z 56.952,A -85,B 0,C 180,E1 24986.067,E2 24986.067} C_VEL
LIN {X 0,Y 520.542,Z 56.953,A -85,B 0,C 180,E1 24982.673,E2 24982.673} C_VEL
LIN {X 0,Y 520.537,Z 56.953,A -85,B 0,C 180,E1 24979.181,E2 24979.181} C_VEL
LIN {X 0,Y 520.579,Z 56.956,A -85,B 0,C 180,E1 24977.869,E2 24977.869} C_VEL
LIN {X 0,Y 519.574,Z 57.084,A -85,B 0,C 180,E1 24977.021,E2 24977.021} C_VEL
LIN {X 0,Y 513.089,Z 57.893,A -85,B 0,C 180,E1 24974.578,E2 24974.578} C_VEL
LIN {X 0,Y 512.644,Z 57.943,A -85,B 0,C 180,E1 24974.019,E2 24974.019} C_VEL
LIN {X 0,Y 512.613,Z 57.944,A -85,B 0,C 180,E1 24970.645,E2 24970.645} C_VEL
LIN {X 0,Y 512.589,Z 57.947,A -85,B 0,C 180,E1 24967.264,E2 24967.264} C_VEL
LIN {X 0,Y 512.643,Z 58.207,A -85,B 0,C 180,E1 24964.822,E2 24964.822} C_VEL
LIN {X 0,Y 515.209,Z 69.499,A -85,B 0,C 180,E1 24963.511,E2 24963.511} C_VEL
LIN {X 0,Y 515.178,Z 100.134,A -85,B 0,C 180,E1 24960.269,E2 24960.269} C_VEL
LIN {X 0,Y 514.899,Z 131.32,A -85,B 0,C 180,E1 24956.9,E2 24956.9} C_VEL
LIN {X 0,Y 514.556,Z 163.182,A -85,B 0,C 180,E1 24953.473,E2 24953.473} C_VEL
LIN {X 0,Y 514.477,Z 182.706,A -85,B 0,C 180,E1 24951.44,E2 24951.44} C_VEL
LIN {X 0,Y 514.977,Z 188.235,A -85,B 0,C 180,E1 24951.34,E2 24951.34} C_VEL
LIN {X 0,Y 514.439,Z 294.324,A -85,B 0,C 180,E1 24949.819,E2 24949.819} C_VEL
LIN {X 0,Y 514.376,Z 308.625,A -85,B 0,C 180,E1 24949.413,E2 24949.413} C_VEL
LIN {X 0,Y 514.207,Z 322.238,A -85,B 0,C 180,E1 24948.83,E2 24948.83} C_VEL
LIN {X 0,Y 513.906,Z 335.846,A -85,B 0,C 180,E1 24948.019,E2 24948.019} C_VEL
LIN {X 0,Y 513.599,Z 347.737,A -85,B 0,C 180,E1 24947.085,E2 24947.085} C_VEL
LIN {X 0,Y 513.31,Z 358.379,A -85,B 0,C 180,E1 24946.026,E2 24946.026} C_VEL
LIN {X 0,Y 512.977,Z 368.954,A -85,B 0,C 180,E1 24944.677,E2 24944.677} C_VEL
LIN {X 0,Y 512.718,Z 377.274,A -85,B 0,C 180,E1 24943.303,E2 24943.303} C_VEL
LIN {X 0,Y 512.527,Z 384.164,A -85,B 0,C 180,E1 24941.819,E2 24941.819} C_VEL
LIN {X 0,Y 512.402,Z 389.535,A -85,B 0,C 180,E1 24940.227,E2 24940.227} C_VEL
LIN {X 0,Y 512.315,Z 393.229,A -85,B 0,C 180,E1 24938.529,E2 24938.529} C_VEL
LIN {X 0,Y 512.277,Z 395.037,A -85,B 0,C 180,E1 24936.837,E2 24936.837} C_VEL
LIN {X 0,Y 512.273,Z 395.072,A -85,B 0,C 180,E1 24935.15,E2 24935.15} C_VEL
LIN {X 0,Y 512.306,Z 393.348,A -85,B 0,C 180,E1 24933.468,E2 24933.468} C_VEL
LIN {X 0,Y 512.393,Z 389.468,A -85,B 0,C 180,E1 24931.676,E2 24931.676} C_VEL
LIN {X 0,Y 512.528,Z 383.736,A -85,B 0,C 180,E1 24929.999,E2 24929.999} C_VEL
LIN {X 0,Y 512.716,Z 376.866,A -85,B 0,C 180,E1 24928.546,E2 24928.546} C_VEL
LIN {X 0,Y 512.969,Z 368.665,A -85,B 0,C 180,E1 24927.206,E2 24927.206} C_VEL
LIN {X 0,Y 513.296,Z 358.097,A -85,B 0,C 180,E1 24925.866,E2 24925.866} C_VEL
LIN {X 0,Y 513.619,Z 346.131,A -85,B 0,C 180,E1 24924.694,E2 24924.694} C_VEL
LIN {X 0,Y 513.942,Z 333.516,A -85,B 0,C 180,E1 24923.745,E2 24923.745} C_VEL
LIN {X 0,Y 514.207,Z 320.901,A -85,B 0,C 180,E1 24923.022,E2 24923.022} C_VEL
LIN {X 0,Y 514.349,Z 306.054,A -85,B 0,C 180,E1 24922.41,E2 24922.41} C_VEL
LIN {X 0,Y 514.398,Z 290.299,A -85,B 0,C 180,E1 24922.013,E2 24922.013} C_VEL
LIN {X 0,Y 514.889,Z 178.871,A -85,B 0,C 180,E1 24920.428,E2 24920.428} C_VEL
LIN {X 0,Y 515.393,Z 125.88,A -85,B 0,C 180,E1 24917.051,E2 24917.051} C_VEL
LIN {X 0,Y 515.879,Z 74.395,A -85,B 0,C 180,E1 24913.735,E2 24913.735} C_VEL
LIN {X 0,Y 515.976,Z 70.334,A -85,B 0,C 180,E1 24913.449,E2 24913.449} C_VEL
LIN {X 0,Y 516.231,Z 69.817,A -85,B 0,C 180,E1 24913.255,E2 24913.255} C_VEL
LIN {X 0,Y 517.538,Z 73.569,A -85,B 0,C 180,E1 24912.865,E2 24912.865} C_VEL
LIN {X 0,Y 516.329,Z 117.686,A -85,B 0,C 180,E1 24909.718,E2 24909.718} C_VEL
LIN {X 0,Y 515.016,Z 168.902,A -85,B 0,C 180,E1 24906.123,E2 24906.123} C_VEL
LIN {X 0,Y 515.078,Z 172.644,A -85,B 0,C 180,E1 24905.916,E2 24905.916} C_VEL
LIN {X 0,Y 515.903,Z 182.691,A -85,B 0,C 180,E1 24905.73,E2 24905.73} C_VEL
LIN {X 0,Y 515,Z 291.045,A -85,B 0,C 180,E1 24904.098,E2 24904.098} C_VEL
LIN {X 0,Y 514.809,Z 306.402,A -85,B 0,C 180,E1 24903.654,E2 24903.654} C_VEL
LIN {X 0,Y 514.484,Z 321.498,A -85,B 0,C 180,E1 24902.982,E2 24902.982} C_VEL
LIN {X 0,Y 514.103,Z 334.7,A -85,B 0,C 180,E1 24902.175,E2 24902.175} C_VEL
LIN {X 0,Y 513.724,Z 347.043,A -85,B 0,C 180,E1 24901.199,E2 24901.199} C_VEL
LIN {X 0,Y 513.322,Z 359.171,A -85,B 0,C 180,E1 24899.961,E2 24899.961} C_VEL
LIN {X 0,Y 512.967,Z 369.354,A -85,B 0,C 180,E1 24898.621,E2 24898.621} C_VEL
LIN {X 0,Y 512.718,Z 377.263,A -85,B 0,C 180,E1 24897.304,E2 24897.304} C_VEL
LIN {X 0,Y 512.508,Z 384.667,A -85,B 0,C 180,E1 24895.68,E2 24895.68} C_VEL
LIN {X 0,Y 512.378,Z 390.003,A -85,B 0,C 180,E1 24894.029,E2 24894.029} C_VEL
LIN {X 0,Y 512.309,Z 393.416,A -85,B 0,C 180,E1 24892.409,E2 24892.409} C_VEL
LIN {X 0,Y 512.285,Z 395.228,A -85,B 0,C 180,E1 24890.616,E2 24890.616} C_VEL
LIN {X 0,Y 512.295,Z 395.048,A -85,B 0,C 180,E1 24888.873,E2 24888.873} C_VEL
LIN {X 0,Y 512.349,Z 393.119,A -85,B 0,C 180,E1 24887.204,E2 24887.204} C_VEL
LIN {X 0,Y 512.45,Z 389.401,A -85,B 0,C 180,E1 24885.536,E2 24885.536} C_VEL
LIN {X 0,Y 512.598,Z 384.038,A -85,B 0,C 180,E1 24883.965,E2 24883.965} C_VEL
LIN {X 0,Y 512.818,Z 377.394,A -85,B 0,C 180,E1 24882.523,E2 24882.523} C_VEL
LIN {X 0,Y 513.136,Z 368.424,A -85,B 0,C 180,E1 24881.046,E2 24881.046} C_VEL
LIN {X 0,Y 513.495,Z 358.69,A -85,B 0,C 180,E1 24879.797,E2 24879.797} C_VEL
LIN {X 0,Y 513.901,Z 347.435,A -85,B 0,C 180,E1 24878.649,E2 24878.649} C_VEL
LIN {X 0,Y 514.354,Z 333.952,A -85,B 0,C 180,E1 24877.589,E2 24877.589} C_VEL
LIN {X 0,Y 514.724,Z 320.559,A -85,B 0,C 180,E1 24876.792,E2 24876.792} C_VEL
LIN {X 0,Y 515.042,Z 306.126,A -85,B 0,C 180,E1 24876.161,E2 24876.161} C_VEL
LIN {X 0,Y 515.26,Z 290.22,A -85,B 0,C 180,E1 24875.709,E2 24875.709} C_VEL
LIN {X 0,Y 516.113,Z 185.054,A -85,B 0,C 180,E1 24874.064,E2 24874.064} C_VEL
LIN {X 0,Y 514.292,Z 174.672,A -85,B 0,C 180,E1 24873.782,E2 24873.782} C_VEL
LIN {X 0,Y 515.227,Z 144.346,A -85,B 0,C 180,E1 24870.174,E2 24870.174} C_VEL
LIN {X 0,Y 516.327,Z 114.921,A -85,B 0,C 180,E1 24866.607,E2 24866.607} C_VEL
LIN {X 0,Y 517.538,Z 85.882,A -85,B 0,C 180,E1 24863.031,E2 24863.031} C_VEL
LIN {X 0,Y 517.858,Z 76.693,A -85,B 0,C 180,E1 24861.879,E2 24861.879} C_VEL
LIN {X 0,Y 513.098,Z 59.867,A -85,B 0,C 180,E1 24859.346,E2 24859.346} C_VEL
LIN {X 0,Y 512.616,Z 58.044,A -85,B 0,C 180,E1 24859.01,E2 24859.01} C_VEL
LIN {X 0,Y 512.624,Z 57.944,A -85,B 0,C 180,E1 24855.615,E2 24855.615} C_VEL
LIN {X 0,Y 512.651,Z 57.943,A -85,B 0,C 180,E1 24852.16,E2 24852.16} C_VEL
LIN {X 0,Y 512.609,Z 57.939,A -85,B 0,C 180,E1 24848.751,E2 24848.751} C_VEL
LIN {X 0,Y 512.595,Z 57.945,A -85,B 0,C 180,E1 24845.373,E2 24845.373} C_VEL
LIN {X 0,Y 512.63,Z 57.945,A -85,B 0,C 180,E1 24842.012,E2 24842.012} C_VEL
LIN {X 0,Y 512.631,Z 57.941,A -85,B 0,C 180,E1 24838.659,E2 24838.659} C_VEL
LIN {X 0,Y 512.592,Z 57.944,A -85,B 0,C 180,E1 24835.301,E2 24835.301} C_VEL
LIN {X 0,Y 512.596,Z 57.945,A -85,B 0,C 180,E1 24831.814,E2 24831.814} C_VEL
LIN {X 0,Y 512.634,Z 57.943,A -85,B 0,C 180,E1 24828.411,E2 24828.411} C_VEL
LIN {X 0,Y 512.621,Z 57.942,A -85,B 0,C 180,E1 24824.965,E2 24824.965} C_VEL
LIN {X 0,Y 512.586,Z 57.942,A -85,B 0,C 180,E1 24821.579,E2 24821.579} C_VEL
LIN {X 0,Y 512.588,Z 57.945,A -85,B 0,C 180,E1 24818.126,E2 24818.126} C_VEL
LIN {X 0,Y 512.638,Z 57.943,A -85,B 0,C 180,E1 24814.822,E2 24814.822} C_VEL
LIN {X 0,Y 512.603,Z 57.945,A -85,B 0,C 180,E1 24811.372,E2 24811.372} C_VEL
LIN {X 0,Y 512.575,Z 57.946,A -85,B 0,C 180,E1 24808.053,E2 24808.053} C_VEL
LIN {X 0,Y 512.607,Z 57.946,A -85,B 0,C 180,E1 24804.735,E2 24804.735} C_VEL
LIN {X 0,Y 512.627,Z 57.946,A -85,B 0,C 180,E1 24801.278,E2 24801.278} C_VEL
LIN {X 0,Y 512.571,Z 57.948,A -85,B 0,C 180,E1 24798.004,E2 24798.004} C_VEL
LIN {X 0,Y 512.575,Z 57.947,A -85,B 0,C 180,E1 24794.444,E2 24794.444} C_VEL
LIN {X 0,Y 512.616,Z 57.944,A -85,B 0,C 180,E1 24791.096,E2 24791.096} C_VEL
LIN {X 0,Y 512.605,Z 57.945,A -85,B 0,C 180,E1 24787.769,E2 24787.769} C_VEL
LIN {X 0,Y 512.609,Z 58.16,A -85,B 0,C 180,E1 24784.637,E2 24784.637} C_VEL
LIN {X 0,Y 514.781,Z 64.242,A -85,B 0,C 180,E1 24783.879,E2 24783.879} C_VEL
LIN {X 0,Y 519.933,Z 79.492,A -85,B 0,C 180,E1 24782.187,E2 24782.187} C_VEL
LIN {X 0,Y 518.005,Z 123.19,A -85,B 0,C 180,E1 24778.663,E2 24778.663} C_VEL
LIN {X 0,Y 516.82,Z 159.261,A -85,B 0,C 180,E1 24775.878,E2 24775.878} C_VEL
LIN {X 0,Y 518.175,Z 171.902,A -85,B 0,C 180,E1 24775.635,E2 24775.635} C_VEL
LIN {X 0,Y 517.061,Z 363.934,A -85,B 0,C 180,E1 24772.929,E2 24772.929} C_VEL
LIN {X 0,Y 516.63,Z 382.746,A -85,B 0,C 180,E1 24772.463,E2 24772.463} C_VEL
LIN {X 0,Y 516.137,Z 400.253,A -85,B 0,C 180,E1 24771.836,E2 24771.836} C_VEL
LIN {X 0,Y 515.574,Z 417.391,A -85,B 0,C 180,E1 24771.025,E2 24771.025} C_VEL
LIN {X 0,Y 514.933,Z 434.77,A -85,B 0,C 180,E1 24769.983,E2 24769.983} C_VEL
LIN {X 0,Y 514.296,Z 451.09,A -85,B 0,C 180,E1 24768.775,E2 24768.775} C_VEL
LIN {X 0,Y 513.711,Z 466.452,A -85,B 0,C 180,E1 24767.395,E2 24767.395} C_VEL
LIN {X 0,Y 513.183,Z 480.935,A -85,B 0,C 180,E1 24765.83,E2 24765.83} C_VEL
LIN {X 0,Y 512.753,Z 494.153,A -85,B 0,C 180,E1 24764.108,E2 24764.108} C_VEL
LIN {X 0,Y 512.448,Z 505.078,A -85,B 0,C 180,E1 24762.394,E2 24762.394} C_VEL
LIN {X 0,Y 512.231,Z 514.65,A -85,B 0,C 180,E1 24760.574,E2 24760.574} C_VEL
LIN {X 0,Y 512.103,Z 522.8,A -85,B 0,C 180,E1 24758.647,E2 24758.647} C_VEL
LIN {X 0,Y 512.022,Z 529.425,A -85,B 0,C 180,E1 24756.617,E2 24756.617} C_VEL
LIN {X 0,Y 511.997,Z 534.167,A -85,B 0,C 180,E1 24754.593,E2 24754.593} C_VEL
LIN {X 0,Y 511.992,Z 537.149,A -85,B 0,C 180,E1 24752.575,E2 24752.575} C_VEL
LIN {X 0,Y 511.994,Z 538.447,A -85,B 0,C 180,E1 24750.56,E2 24750.56} C_VEL
LIN {X 0,Y 511.993,Z 538.018,A -85,B 0,C 180,E1 24748.434,E2 24748.434} C_VEL
LIN {X 0,Y 511.988,Z 535.732,A -85,B 0,C 180,E1 24746.306,E2 24746.306} C_VEL
LIN {X 0,Y 512.003,Z 531.802,A -85,B 0,C 180,E1 24744.285,E2 24744.285} C_VEL
LIN {X 0,Y 512.061,Z 526.061,A -85,B 0,C 180,E1 24742.258,E2 24742.258} C_VEL
LIN {X 0,Y 512.152,Z 518.842,A -85,B 0,C 180,E1 24740.336,E2 24740.336} C_VEL
LIN {X 0,Y 512.333,Z 509.676,A -85,B 0,C 180,E1 24738.405,E2 24738.405} C_VEL
LIN {X 0,Y 512.628,Z 499.002,A -85,B 0,C 180,E1 24736.58,E2 24736.58} C_VEL
LIN {X 0,Y 512.999,Z 486.846,A -85,B 0,C 180,E1 24734.862,E2 24734.862} C_VEL
LIN {X 0,Y 513.498,Z 473.173,A -85,B 0,C 180,E1 24733.252,E2 24733.252} C_VEL
LIN {X 0,Y 514.063,Z 458.479,A -85,B 0,C 180,E1 24731.811,E2 24731.811} C_VEL
LIN {X 0,Y 514.69,Z 442.8,A -85,B 0,C 180,E1 24730.534,E2 24730.534} C_VEL
LIN {X 0,Y 515.33,Z 426.443,A -85,B 0,C 180,E1 24729.442,E2 24729.442} C_VEL
LIN {X 0,Y 515.981,Z 408.524,A -85,B 0,C 180,E1 24728.482,E2 24728.482} C_VEL
LIN {X 0,Y 516.57,Z 389.722,A -85,B 0,C 180,E1 24727.718,E2 24727.718} C_VEL
LIN {X 0,Y 517.037,Z 370.75,A -85,B 0,C 180,E1 24727.173,E2 24727.173} C_VEL
LIN {X 0,Y 517.322,Z 350.11,A -85,B 0,C 180,E1 24726.81,E2 24726.81} C_VEL
LIN {X 0,Y 518.28,Z 162.067,A -85,B 0,C 180,E1 24724.159,E2 24724.159} C_VEL
LIN {X 0,Y 517.878,Z 154.885,A -85,B 0,C 180,E1 24724.008,E2 24724.008} C_VEL
LIN {X 0,Y 519.873,Z 77.623,A -85,B 0,C 180,E1 24720.442,E2 24720.442} C_VEL
LIN {X 0,Y 512.712,Z 58.424,A -85,B 0,C 180,E1 24719.07,E2 24719.07} C_VEL
LIN {X 0,Y 512.637,Z 57.945,A -85,B 0,C 180,E1 24718.88,E2 24718.88} C_VEL
LIN {X 0,Y 512.635,Z 57.942,A -85,B 0,C 180,E1 24715.285,E2 24715.285} C_VEL
LIN {X 0,Y 512.647,Z 57.942,A -85,B 0,C 180,E1 24711.812,E2 24711.812} C_VEL
LIN {X 0,Y 512.641,Z 57.941,A -85,B 0,C 180,E1 24708.313,E2 24708.313} C_VEL
LIN {X 0,Y 512.646,Z 57.937,A -85,B 0,C 180,E1 24704.756,E2 24704.756} C_VEL
LIN {X 0,Y 512.631,Z 57.937,A -85,B 0,C 180,E1 24701.243,E2 24701.243} C_VEL
LIN {X 0,Y 512.634,Z 57.943,A -85,B 0,C 180,E1 24697.766,E2 24697.766} C_VEL
LIN {X 0,Y 512.648,Z 57.941,A -85,B 0,C 180,E1 24694.215,E2 24694.215} C_VEL
LIN {X 0,Y 512.646,Z 57.937,A -85,B 0,C 180,E1 24690.673,E2 24690.673} C_VEL
LIN {X 0,Y 512.64,Z 57.934,A -85,B 0,C 180,E1 24687.155,E2 24687.155} C_VEL
LIN {X 0,Y 512.622,Z 57.935,A -85,B 0,C 180,E1 24683.691,E2 24683.691} C_VEL
LIN {X 0,Y 512.63,Z 57.94,A -85,B 0,C 180,E1 24680.196,E2 24680.196} C_VEL
LIN {X 0,Y 512.649,Z 57.941,A -85,B 0,C 180,E1 24676.744,E2 24676.744} C_VEL
LIN {X 0,Y 512.648,Z 57.934,A -85,B 0,C 180,E1 24673.191,E2 24673.191} C_VEL
LIN {X 0,Y 512.621,Z 57.934,A -85,B 0,C 180,E1 24669.77,E2 24669.77} C_VEL
LIN {X 0,Y 512.618,Z 57.94,A -85,B 0,C 180,E1 24666.271,E2 24666.271} C_VEL
LIN {X 0,Y 512.64,Z 57.944,A -85,B 0,C 180,E1 24662.795,E2 24662.795} C_VEL
LIN {X 0,Y 512.651,Z 57.933,A -85,B 0,C 180,E1 24659.329,E2 24659.329} C_VEL
LIN {X 0,Y 512.626,Z 57.937,A -85,B 0,C 180,E1 24655.861,E2 24655.861} C_VEL
LIN {X 0,Y 512.609,Z 57.941,A -85,B 0,C 180,E1 24652.378,E2 24652.378} C_VEL
LIN {X 0,Y 512.631,Z 57.944,A -85,B 0,C 180,E1 24648.98,E2 24648.98} C_VEL
LIN {X 0,Y 512.653,Z 57.935,A -85,B 0,C 180,E1 24645.543,E2 24645.543} C_VEL
LIN {X 0,Y 512.625,Z 57.936,A -85,B 0,C 180,E1 24642.05,E2 24642.05} C_VEL
LIN {X 0,Y 512.604,Z 57.939,A -85,B 0,C 180,E1 24638.607,E2 24638.607} C_VEL
LIN {X 0,Y 512.622,Z 57.937,A -85,B 0,C 180,E1 24635.206,E2 24635.206} C_VEL
LIN {X 0,Y 512.651,Z 57.941,A -85,B 0,C 180,E1 24631.709,E2 24631.709} C_VEL
LIN {X 0,Y 512.625,Z 57.936,A -85,B 0,C 180,E1 24628.252,E2 24628.252} C_VEL
LIN {X 0,Y 512.599,Z 57.936,A -85,B 0,C 180,E1 24624.811,E2 24624.811} C_VEL
LIN {X 0,Y 512.602,Z 57.943,A -85,B 0,C 180,E1 24621.278,E2 24621.278} C_VEL
LIN {X 0,Y 512.641,Z 57.945,A -85,B 0,C 180,E1 24617.86,E2 24617.86} C_VEL
LIN {X 0,Y 512.628,Z 57.942,A -85,B 0,C 180,E1 24614.442,E2 24614.442} C_VEL
LIN {X 0,Y 512.644,Z 57.943,A -85,B 0,C 180,E1 24614.019,E2 24614.019} C_VEL
LIN {X 0,Y 511.657,Z 58.061,A -85,B 0,C 180,E1 24613.159,E2 24613.159} C_VEL
LIN {X 0,Y 505.184,Z 58.869,A -85,B 0,C 180,E1 24610.677,E2 24610.677} C_VEL
LIN {X 0,Y 504.709,Z 58.928,A -85,B 0,C 180,E1 24610.11,E2 24610.11} C_VEL
LIN {X 0,Y 504.682,Z 58.934,A -85,B 0,C 180,E1 24606.606,E2 24606.606} C_VEL
LIN {X 0,Y 504.683,Z 59.161,A -85,B 0,C 180,E1 24605.135,E2 24605.135} C_VEL
LIN {X 0,Y 507.596,Z 71.546,A -85,B 0,C 180,E1 24603.674,E2 24603.674} C_VEL
LIN {X 0,Y 507.521,Z 102.744,A -85,B 0,C 180,E1 24600.356,E2 24600.356} C_VEL
LIN {X 0,Y 507.228,Z 133.7,A -85,B 0,C 180,E1 24597.001,E2 24597.001} C_VEL
LIN {X 0,Y 506.857,Z 166.529,A -85,B 0,C 180,E1 24593.466,E2 24593.466} C_VEL
LIN {X 0,Y 506.813,Z 183.687,A -85,B 0,C 180,E1 24591.688,E2 24591.688} C_VEL
LIN {X 0,Y 507.311,Z 189.125,A -85,B 0,C 180,E1 24591.587,E2 24591.587} C_VEL
LIN {X 0,Y 506.725,Z 295.427,A -85,B 0,C 180,E1 24590.037,E2 24590.037} C_VEL
LIN {X 0,Y 506.66,Z 309.867,A -85,B 0,C 180,E1 24589.619,E2 24589.619} C_VEL
LIN {X 0,Y 506.473,Z 323.779,A -85,B 0,C 180,E1 24589.009,E2 24589.009} C_VEL
LIN {X 0,Y 506.144,Z 337.673,A -85,B 0,C 180,E1 24588.159,E2 24588.159} C_VEL
LIN {X 0,Y 505.792,Z 350.272,A -85,B 0,C 180,E1 24587.129,E2 24587.129} C_VEL
LIN {X 0,Y 505.441,Z 361.379,A -85,B 0,C 180,E1 24585.959,E2 24585.959} C_VEL
LIN {X 0,Y 505.111,Z 370.963,A -85,B 0,C 180,E1 24584.676,E2 24584.676} C_VEL
LIN {X 0,Y 504.82,Z 379.696,A -85,B 0,C 180,E1 24583.165,E2 24583.165} C_VEL
LIN {X 0,Y 504.604,Z 386.669,A -85,B 0,C 180,E1 24581.543,E2 24581.543} C_VEL
LIN {X 0,Y 504.466,Z 391.596,A -85,B 0,C 180,E1 24579.914,E2 24579.914} C_VEL
LIN {X 0,Y 504.388,Z 394.697,A -85,B 0,C 180,E1 24578.319,E2 24578.319} C_VEL
LIN {X 0,Y 504.351,Z 396.268,A -85,B 0,C 180,E1 24576.602,E2 24576.602} C_VEL
LIN {X 0,Y 504.354,Z 395.953,A -85,B 0,C 180,E1 24574.775,E2 24574.775} C_VEL
LIN {X 0,Y 504.399,Z 393.813,A -85,B 0,C 180,E1 24573.067,E2 24573.067} C_VEL
LIN {X 0,Y 504.497,Z 390.167,A -85,B 0,C 180,E1 24571.475,E2 24571.475} C_VEL
LIN {X 0,Y 504.645,Z 384.742,A -85,B 0,C 180,E1 24569.886,E2 24569.886} C_VEL
LIN {X 0,Y 504.878,Z 377.234,A -85,B 0,C 180,E1 24568.297,E2 24568.297} C_VEL
LIN {X 0,Y 505.162,Z 368.794,A -85,B 0,C 180,E1 24566.936,E2 24566.936} C_VEL
LIN {X 0,Y 505.512,Z 358.453,A -85,B 0,C 180,E1 24565.632,E2 24565.632} C_VEL
LIN {X 0,Y 505.85,Z 346.95,A -85,B 0,C 180,E1 24564.498,E2 24564.498} C_VEL
LIN {X 0,Y 506.195,Z 334.236,A -85,B 0,C 180,E1 24563.535,E2 24563.535} C_VEL
LIN {X 0,Y 506.473,Z 321.403,A -85,B 0,C 180,E1 24562.798,E2 24562.798} C_VEL
LIN {X 0,Y 506.615,Z 306.841,A -85,B 0,C 180,E1 24562.196,E2 24562.196} C_VEL
LIN {X 0,Y 506.658,Z 291.103,A -85,B 0,C 180,E1 24561.797,E2 24561.797} C_VEL
LIN {X 0,Y 507.216,Z 179.658,A -85,B 0,C 180,E1 24560.187,E2 24560.187} C_VEL
LIN {X 0,Y 507.734,Z 126.484,A -85,B 0,C 180,E1 24556.794,E2 24556.794} C_VEL
LIN {X 0,Y 508.303,Z 75.674,A -85,B 0,C 180,E1 24553.486,E2 24553.486} C_VEL
LIN {X 0,Y 508.771,Z 74.885,A -85,B 0,C 180,E1 24553.296,E2 24553.296} C_VEL
LIN {X 0,Y 510.102,Z 76.042,A -85,B 0,C 180,E1 24553.077,E2 24553.077} C_VEL
LIN {X 0,Y 508.702,Z 122.078,A -85,B 0,C 180,E1 24549.761,E2 24549.761} C_VEL
LIN {X 0,Y 507.374,Z 171.767,A -85,B 0,C 180,E1 24546.249,E2 24546.249} C_VEL
LIN {X 0,Y 508.367,Z 183.332,A -85,B 0,C 180,E1 24546.025,E2 24546.025} C_VEL
LIN {X 0,Y 507.37,Z 291.618,A -85,B 0,C 180,E1 24544.36,E2 24544.36} C_VEL
LIN {X 0,Y 507.168,Z 306.704,A -85,B 0,C 180,E1 24543.919,E2 24543.919} C_VEL
LIN {X 0,Y 506.828,Z 321.289,A -85,B 0,C 180,E1 24543.269,E2 24543.269} C_VEL
LIN {X 0,Y 506.436,Z 334.278,A -85,B 0,C 180,E1 24542.484,E2 24542.484} C_VEL
LIN {X 0,Y 505.987,Z 347.594,A -85,B 0,C 180,E1 24541.431,E2 24541.431} C_VEL
LIN {X 0,Y 505.56,Z 359.246,A -85,B 0,C 180,E1 24540.237,E2 24540.237} C_VEL
LIN {X 0,Y 505.192,Z 368.96,A -85,B 0,C 180,E1 24538.98,E2 24538.98} C_VEL
LIN {X 0,Y 504.879,Z 377.78,A -85,B 0,C 180,E1 24537.528,E2 24537.528} C_VEL
LIN {X 0,Y 504.633,Z 385.17,A -85,B 0,C 180,E1 24535.916,E2 24535.916} C_VEL
LIN {X 0,Y 504.49,Z 390.407,A -85,B 0,C 180,E1 24534.35,E2 24534.35} C_VEL
LIN {X 0,Y 504.402,Z 394.207,A -85,B 0,C 180,E1 24532.645,E2 24532.645} C_VEL
LIN {X 0,Y 504.36,Z 396.153,A -85,B 0,C 180,E1 24530.919,E2 24530.919} C_VEL
LIN {X 0,Y 504.371,Z 396.362,A -85,B 0,C 180,E1 24529.225,E2 24529.225} C_VEL
LIN {X 0,Y 504.42,Z 394.745,A -85,B 0,C 180,E1 24527.473,E2 24527.473} C_VEL
LIN {X 0,Y 504.523,Z 391.513,A -85,B 0,C 180,E1 24525.841,E2 24525.841} C_VEL
LIN {X 0,Y 504.691,Z 386.406,A -85,B 0,C 180,E1 24524.179,E2 24524.179} C_VEL
LIN {X 0,Y 504.943,Z 379.339,A -85,B 0,C 180,E1 24522.556,E2 24522.556} C_VEL
LIN {X 0,Y 505.263,Z 371.208,A -85,B 0,C 180,E1 24521.142,E2 24521.142} C_VEL
LIN {X 0,Y 505.676,Z 361.333,A -85,B 0,C 180,E1 24519.795,E2 24519.795} C_VEL
LIN {X 0,Y 506.142,Z 349.397,A -85,B 0,C 180,E1 24518.53,E2 24518.53} C_VEL
LIN {X 0,Y 506.575,Z 338.01,A -85,B 0,C 180,E1 24517.582,E2 24517.582} C_VEL
LIN {X 0,Y 507.019,Z 324.283,A -85,B 0,C 180,E1 24516.693,E2 24516.693} C_VEL
LIN {X 0,Y 507.378,Z 309.624,A -85,B 0,C 180,E1 24516.001,E2 24516.001} C_VEL
LIN {X 0,Y 507.625,Z 294.824,A -85,B 0,C 180,E1 24515.525,E2 24515.525} C_VEL
LIN {X 0,Y 507.875,Z 271.586,A -85,B 0,C 180,E1 24515.109,E2 24515.109} C_VEL
LIN {X 0,Y 508.668,Z 186.225,A -85,B 0,C 180,E1 24513.753,E2 24513.753} C_VEL
LIN {X 0,Y 506.603,Z 174.554,A -85,B 0,C 180,E1 24513.429,E2 24513.429} C_VEL
LIN {X 0,Y 507.624,Z 144.69,A -85,B 0,C 180,E1 24509.825,E2 24509.825} C_VEL
LIN {X 0,Y 508.784,Z 116.325,A -85,B 0,C 180,E1 24506.346,E2 24506.346} C_VEL
LIN {X 0,Y 510.126,Z 87.266,A -85,B 0,C 180,E1 24502.714,E2 24502.714} C_VEL
LIN {X 0,Y 510.273,Z 78.708,A -85,B 0,C 180,E1 24501.616,E2 24501.616} C_VEL
LIN {X 0,Y 505.315,Z 61.28,A -85,B 0,C 180,E1 24498.936,E2 24498.936} C_VEL
LIN {X 0,Y 504.696,Z 59.057,A -85,B 0,C 180,E1 24498.54,E2 24498.54} C_VEL
LIN {X 0,Y 504.663,Z 58.932,A -85,B 0,C 180,E1 24495.043,E2 24495.043} C_VEL
LIN {X 0,Y 504.673,Z 58.931,A -85,B 0,C 180,E1 24491.543,E2 24491.543} C_VEL
LIN {X 0,Y 504.711,Z 58.93,A -85,B 0,C 180,E1 24488.086,E2 24488.086} C_VEL
LIN {X 0,Y 504.682,Z 58.932,A -85,B 0,C 180,E1 24484.659,E2 24484.659} C_VEL
LIN {X 0,Y 504.656,Z 58.932,A -85,B 0,C 180,E1 24481.249,E2 24481.249} C_VEL
LIN {X 0,Y 504.661,Z 58.934,A -85,B 0,C 180,E1 24477.729,E2 24477.729} C_VEL
LIN {X 0,Y 504.701,Z 58.932,A -85,B 0,C 180,E1 24474.315,E2 24474.315} C_VEL
LIN {X 0,Y 504.681,Z 58.932,A -85,B 0,C 180,E1 24470.881,E2 24470.881} C_VEL
LIN {X 0,Y 504.648,Z 58.933,A -85,B 0,C 180,E1 24467.528,E2 24467.528} C_VEL
LIN {X 0,Y 504.654,Z 58.932,A -85,B 0,C 180,E1 24464.014,E2 24464.014} C_VEL
LIN {X 0,Y 504.692,Z 58.933,A -85,B 0,C 180,E1 24460.564,E2 24460.564} C_VEL
LIN {X 0,Y 504.678,Z 58.932,A -85,B 0,C 180,E1 24457.109,E2 24457.109} C_VEL
LIN {X 0,Y 504.642,Z 58.934,A -85,B 0,C 180,E1 24453.779,E2 24453.779} C_VEL
LIN {X 0,Y 504.648,Z 58.935,A -85,B 0,C 180,E1 24450.309,E2 24450.309} C_VEL
LIN {X 0,Y 504.691,Z 58.934,A -85,B 0,C 180,E1 24446.931,E2 24446.931} C_VEL
LIN {X 0,Y 504.657,Z 58.934,A -85,B 0,C 180,E1 24443.532,E2 24443.532} C_VEL
LIN {X 0,Y 504.632,Z 58.937,A -85,B 0,C 180,E1 24440.21,E2 24440.21} C_VEL
LIN {X 0,Y 504.657,Z 58.934,A -85,B 0,C 180,E1 24436.812,E2 24436.812} C_VEL
LIN {X 0,Y 504.691,Z 58.93,A -85,B 0,C 180,E1 24433.358,E2 24433.358} C_VEL
LIN {X 0,Y 504.642,Z 58.938,A -85,B 0,C 180,E1 24430.086,E2 24430.086} C_VEL
LIN {X 0,Y 504.641,Z 58.939,A -85,B 0,C 180,E1 24426.611,E2 24426.611} C_VEL
LIN {X 0,Y 504.701,Z 59.137,A -85,B 0,C 180,E1 24425.148,E2 24425.148} C_VEL
LIN {X 0,Y 507.036,Z 65.951,A -85,B 0,C 180,E1 24424.284,E2 24424.284} C_VEL
LIN {X 0,Y 512.633,Z 82.144,A -85,B 0,C 180,E1 24422.437,E2 24422.437} C_VEL
LIN {X 0,Y 510.555,Z 124.282,A -85,B 0,C 180,E1 24418.97,E2 24418.97} C_VEL
LIN {X 0,Y 509.256,Z 159.474,A -85,B 0,C 180,E1 24416.2,E2 24416.2} C_VEL
LIN {X 0,Y 510.684,Z 172.821,A -85,B 0,C 180,E1 24415.939,E2 24415.939} C_VEL
LIN {X 0,Y 509.458,Z 363.311,A -85,B 0,C 180,E1 24413.219,E2 24413.219} C_VEL
LIN {X 0,Y 508.993,Z 382.07,A -85,B 0,C 180,E1 24412.748,E2 24412.748} C_VEL
LIN {X 0,Y 508.441,Z 400.023,A -85,B 0,C 180,E1 24412.093,E2 24412.093} C_VEL
LIN {X 0,Y 507.801,Z 417.558,A -85,B 0,C 180,E1 24411.242,E2 24411.242} C_VEL
LIN {X 0,Y 507.107,Z 434.731,A -85,B 0,C 180,E1 24410.185,E2 24410.185} C_VEL
LIN {X 0,Y 506.422,Z 450.829,A -85,B 0,C 180,E1 24408.965,E2 24408.965} C_VEL
LIN {X 0,Y 505.762,Z 466.832,A -85,B 0,C 180,E1 24407.488,E2 24407.488} C_VEL
LIN {X 0,Y 505.227,Z 480.514,A -85,B 0,C 180,E1 24405.968,E2 24405.968} C_VEL
LIN {X 0,Y 504.775,Z 493.635,A -85,B 0,C 180,E1 24404.219,E2 24404.219} C_VEL
LIN {X 0,Y 504.465,Z 504.474,A -85,B 0,C 180,E1 24402.477,E2 24402.477} C_VEL
LIN {X 0,Y 504.247,Z 513.964,A -85,B 0,C 180,E1 24400.627,E2 24400.627} C_VEL
LIN {X 0,Y 504.13,Z 522.037,A -85,B 0,C 180,E1 24398.67,E2 24398.67} C_VEL
LIN {X 0,Y 504.072,Z 528.265,A -85,B 0,C 180,E1 24396.721,E2 24396.721} C_VEL
LIN {X 0,Y 504.059,Z 533.03,A -85,B 0,C 180,E1 24394.666,E2 24394.666} C_VEL
LIN {X 0,Y 504.064,Z 536.03,A -85,B 0,C 180,E1 24392.616,E2 24392.616} C_VEL
LIN {X 0,Y 504.072,Z 537.34,A -85,B 0,C 180,E1 24390.569,E2 24390.569} C_VEL
LIN {X 0,Y 504.066,Z 536.915,A -85,B 0,C 180,E1 24388.41,E2 24388.41} C_VEL
LIN {X 0,Y 504.051,Z 534.795,A -85,B 0,C 180,E1 24386.362,E2 24386.362} C_VEL
LIN {X 0,Y 504.05,Z 530.955,A -85,B 0,C 180,E1 24384.309,E2 24384.309} C_VEL
LIN {X 0,Y 504.092,Z 525.302,A -85,B 0,C 180,E1 24382.25,E2 24382.25} C_VEL
LIN {X 0,Y 504.181,Z 517.689,A -85,B 0,C 180,E1 24380.181,E2 24380.181} C_VEL
LIN {X 0,Y 504.361,Z 508.497,A -85,B 0,C 180,E1 24378.219,E2 24378.219} C_VEL
LIN {X 0,Y 504.663,Z 497.789,A -85,B 0,C 180,E1 24376.364,E2 24376.364} C_VEL
LIN {X 0,Y 505.069,Z 485.442,A -85,B 0,C 180,E1 24374.598,E2 24374.598} C_VEL
LIN {X 0,Y 505.607,Z 471.859,A -85,B 0,C 180,E1 24372.983,E2 24372.983} C_VEL
LIN {X 0,Y 506.228,Z 457.09,A -85,B 0,C 180,E1 24371.519,E2 24371.519} C_VEL
LIN {X 0,Y 506.951,Z 440.617,A -85,B 0,C 180,E1 24370.171,E2 24370.171} C_VEL
LIN {X 0,Y 507.663,Z 423.827,A -85,B 0,C 180,E1 24369.056,E2 24369.056} C_VEL
LIN {X 0,Y 508.359,Z 406.031,A -85,B 0,C 180,E1 24368.118,E2 24368.118} C_VEL
LIN {X 0,Y 508.985,Z 387.606,A -85,B 0,C 180,E1 24367.38,E2 24367.38} C_VEL
LIN {X 0,Y 509.479,Z 369.146,A -85,B 0,C 180,E1 24366.857,E2 24366.857} C_VEL
LIN {X 0,Y 509.766,Z 347.602,A -85,B 0,C 180,E1 24366.484,E2 24366.484} C_VEL
LIN {X 0,Y 510.807,Z 162.668,A -85,B 0,C 180,E1 24363.845,E2 24363.845} C_VEL
LIN {X 0,Y 510.377,Z 155.148,A -85,B 0,C 180,E1 24363.691,E2 24363.691} C_VEL
LIN {X 0,Y 512.554,Z 79.563,A -85,B 0,C 180,E1 24360.139,E2 24360.139} C_VEL
LIN {X 0,Y 504.8,Z 59.51,A -85,B 0,C 180,E1 24358.663,E2 24358.663} C_VEL
LIN {X 0,Y 504.707,Z 58.926,A -85,B 0,C 180,E1 24358.414,E2 24358.414} C_VEL
LIN {X 0,Y 504.699,Z 58.928,A -85,B 0,C 180,E1 24354.904,E2 24354.904} C_VEL
LIN {X 0,Y 504.695,Z 58.932,A -85,B 0,C 180,E1 24351.312,E2 24351.312} C_VEL
LIN {X 0,Y 504.707,Z 58.931,A -85,B 0,C 180,E1 24347.81,E2 24347.81} C_VEL
LIN {X 0,Y 504.704,Z 58.931,A -85,B 0,C 180,E1 24344.214,E2 24344.214} C_VEL
LIN {X 0,Y 504.709,Z 58.924,A -85,B 0,C 180,E1 24340.649,E2 24340.649} C_VEL
LIN {X 0,Y 504.694,Z 58.928,A -85,B 0,C 180,E1 24337.174,E2 24337.174} C_VEL
LIN {X 0,Y 504.689,Z 58.93,A -85,B 0,C 180,E1 24333.69,E2 24333.69} C_VEL
LIN {X 0,Y 504.71,Z 58.932,A -85,B 0,C 180,E1 24330.211,E2 24330.211} C_VEL
LIN {X 0,Y 504.706,Z 58.926,A -85,B 0,C 180,E1 24326.692,E2 24326.692} C_VEL
LIN {X 0,Y 504.708,Z 58.921,A -85,B 0,C 180,E1 24323.094,E2 24323.094} C_VEL
LIN {X 0,Y 504.682,Z 58.925,A -85,B 0,C 180,E1 24319.682,E2 24319.682} C_VEL
LIN {X 0,Y 504.683,Z 58.929,A -85,B 0,C 180,E1 24316.089,E2 24316.089} C_VEL
LIN {X 0,Y 504.703,Z 58.932,A -85,B 0,C 180,E1 24312.587,E2 24312.587} C_VEL
LIN {X 0,Y 504.709,Z 58.924,A -85,B 0,C 180,E1 24309.004,E2 24309.004} C_VEL
LIN {X 0,Y 504.703,Z 58.924,A -85,B 0,C 180,E1 24305.456,E2 24305.456} C_VEL
LIN {X 0,Y 504.68,Z 58.928,A -85,B 0,C 180,E1 24301.93,E2 24301.93} C_VEL
LIN {X 0,Y 504.676,Z 58.93,A -85,B 0,C 180,E1 24298.41,E2 24298.41} C_VEL
LIN {X 0,Y 504.694,Z 58.929,A -85,B 0,C 180,E1 24294.885,E2 24294.885} C_VEL
LIN {X 0,Y 504.712,Z 58.928,A -85,B 0,C 180,E1 24291.455,E2 24291.455} C_VEL
LIN {X 0,Y 504.684,Z 58.928,A -85,B 0,C 180,E1 24287.993,E2 24287.993} C_VEL
LIN {X 0,Y 504.668,Z 58.93,A -85,B 0,C 180,E1 24284.604,E2 24284.604} C_VEL
LIN {X 0,Y 504.691,Z 58.933,A -85,B 0,C 180,E1 24281.16,E2 24281.16} C_VEL
LIN {X 0,Y 504.714,Z 58.922,A -85,B 0,C 180,E1 24277.644,E2 24277.644} C_VEL
LIN {X 0,Y 504.694,Z 58.925,A -85,B 0,C 180,E1 24274.079,E2 24274.079} C_VEL
LIN {X 0,Y 504.663,Z 58.923,A -85,B 0,C 180,E1 24270.659,E2 24270.659} C_VEL
LIN {X 0,Y 504.666,Z 58.933,A -85,B 0,C 180,E1 24267.121,E2 24267.121} C_VEL
LIN {X 0,Y 504.694,Z 58.926,A -85,B 0,C 180,E1 24263.675,E2 24263.675} C_VEL
LIN {X 0,Y 504.704,Z 58.928,A -85,B 0,C 180,E1 24260.216,E2 24260.216} C_VEL
LIN {X 0,Y 504.661,Z 58.931,A -85,B 0,C 180,E1 24256.809,E2 24256.809} C_VEL
LIN {X 0,Y 504.655,Z 58.929,A -85,B 0,C 180,E1 24253.274,E2 24253.274} C_VEL
LIN {X 0,Y 504.709,Z 58.928,A -85,B 0,C 180,E1 24250.11,E2 24250.11} C_VEL
LIN {X 0,Y 503.68,Z 59.06,A -85,B 0,C 180,E1 24249.236,E2 24249.236} C_VEL
LIN {X 0,Y 497.222,Z 59.865,A -85,B 0,C 180,E1 24246.715,E2 24246.715} C_VEL
LIN {X 0,Y 496.76,Z 59.922,A -85,B 0,C 180,E1 24246.138,E2 24246.138} C_VEL
LIN {X 0,Y 496.74,Z 60.116,A -85,B 0,C 180,E1 24245.463,E2 24245.463} C_VEL
LIN {X 0,Y 499.973,Z 73.051,A -85,B 0,C 180,E1 24243.908,E2 24243.908} C_VEL
LIN {X 0,Y 499.926,Z 102.684,A -85,B 0,C 180,E1 24240.745,E2 24240.745} C_VEL
LIN {X 0,Y 499.594,Z 134.337,A -85,B 0,C 180,E1 24237.302,E2 24237.302} C_VEL
LIN {X 0,Y 499.21,Z 167.377,A -85,B 0,C 180,E1 24233.738,E2 24233.738} C_VEL
LIN {X 0,Y 499.139,Z 184.441,A -85,B 0,C 180,E1 24231.956,E2 24231.956} C_VEL
LIN {X 0,Y 499.661,Z 189.922,A -85,B 0,C 180,E1 24231.846,E2 24231.846} C_VEL
LIN {X 0,Y 499.031,Z 296.353,A -85,B 0,C 180,E1 24230.272,E2 24230.272} C_VEL
LIN {X 0,Y 498.97,Z 310.781,A -85,B 0,C 180,E1 24229.851,E2 24229.851} C_VEL
LIN {X 0,Y 498.772,Z 324.722,A -85,B 0,C 180,E1 24229.232,E2 24229.232} C_VEL
LIN {X 0,Y 498.414,Z 338.81,A -85,B 0,C 180,E1 24228.357,E2 24228.357} C_VEL
LIN {X 0,Y 498.026,Z 351.685,A -85,B 0,C 180,E1 24227.284,E2 24227.284} C_VEL
LIN {X 0,Y 497.641,Z 362.714,A -85,B 0,C 180,E1 24226.096,E2 24226.096} C_VEL
LIN {X 0,Y 497.279,Z 372.235,A -85,B 0,C 180,E1 24224.793,E2 24224.793} C_VEL
LIN {X 0,Y 496.956,Z 380.919,A -85,B 0,C 180,E1 24223.258,E2 24223.258} C_VEL
LIN {X 0,Y 496.715,Z 387.86,A -85,B 0,C 180,E1 24221.612,E2 24221.612} C_VEL
LIN {X 0,Y 496.551,Z 393.009,A -85,B 0,C 180,E1 24219.854,E2 24219.854} C_VEL
LIN {X 0,Y 496.464,Z 396.129,A -85,B 0,C 180,E1 24218.103,E2 24218.103} C_VEL
LIN {X 0,Y 496.423,Z 397.417,A -85,B 0,C 180,E1 24216.359,E2 24216.359} C_VEL
LIN {X 0,Y 496.433,Z 396.945,A -85,B 0,C 180,E1 24214.62,E2 24214.62} C_VEL
LIN {X 0,Y 496.497,Z 394.46,A -85,B 0,C 180,E1 24212.769,E2 24212.769} C_VEL
LIN {X 0,Y 496.622,Z 390.174,A -85,B 0,C 180,E1 24211.037,E2 24211.037} C_VEL
LIN {X 0,Y 496.807,Z 384.276,A -85,B 0,C 180,E1 24209.423,E2 24209.423} C_VEL
LIN {X 0,Y 497.067,Z 376.906,A -85,B 0,C 180,E1 24207.924,E2 24207.924} C_VEL
LIN {X 0,Y 497.396,Z 368.082,A -85,B 0,C 180,E1 24206.542,E2 24206.542} C_VEL
LIN {X 0,Y 497.786,Z 357.178,A -85,B 0,C 180,E1 24205.218,E2 24205.218} C_VEL
LIN {X 0,Y 498.129,Z 345.635,A -85,B 0,C 180,E1 24204.124,E2 24204.124} C_VEL
LIN {X 0,Y 498.495,Z 333.111,A -85,B 0,C 180,E1 24203.203,E2 24203.203} C_VEL
LIN {X 0,Y 498.772,Z 319.498,A -85,B 0,C 180,E1 24202.454,E2 24202.454} C_VEL
LIN {X 0,Y 498.889,Z 304.717,A -85,B 0,C 180,E1 24201.889,E2 24201.889} C_VEL
LIN {X 0,Y 498.905,Z 289.892,A -85,B 0,C 180,E1 24201.547,E2 24201.547} C_VEL
LIN {X 0,Y 499.547,Z 180.51,A -85,B 0,C 180,E1 24199.945,E2 24199.945} C_VEL
LIN {X 0,Y 500.064,Z 127.929,A -85,B 0,C 180,E1 24196.588,E2 24196.588} C_VEL
LIN {X 0,Y 500.62,Z 81.039,A -85,B 0,C 180,E1 24193.524,E2 24193.524} C_VEL
LIN {X 0,Y 501.069,Z 80.153,A -85,B 0,C 180,E1 24193.33,E2 24193.33} C_VEL
LIN {X 0,Y 502.623,Z 81.041,A -85,B 0,C 180,E1 24193.108,E2 24193.108} C_VEL
LIN {X 0,Y 500.841,Z 133.353,A -85,B 0,C 180,E1 24189.307,E2 24189.307} C_VEL
LIN {X 0,Y 499.778,Z 171.882,A -85,B 0,C 180,E1 24186.566,E2 24186.566} C_VEL
LIN {X 0,Y 500.845,Z 183.97,A -85,B 0,C 180,E1 24186.329,E2 24186.329} C_VEL
LIN {X 0,Y 499.75,Z 292.137,A -85,B 0,C 180,E1 24184.631,E2 24184.631} C_VEL
LIN {X 0,Y 499.525,Z 307.519,A -85,B 0,C 180,E1 24184.173,E2 24184.173} C_VEL
LIN {X 0,Y 499.138,Z 322.948,A -85,B 0,C 180,E1 24183.467,E2 24183.467} C_VEL
LIN {X 0,Y 498.68,Z 336.537,A -85,B 0,C 180,E1 24182.609,E2 24182.609} C_VEL
LIN {X 0,Y 498.227,Z 348.892,A -85,B 0,C 180,E1 24181.6,E2 24181.6} C_VEL
LIN {X 0,Y 497.745,Z 361.093,A -85,B 0,C 180,E1 24180.317,E2 24180.317} C_VEL
LIN {X 0,Y 497.311,Z 371.367,A -85,B 0,C 180,E1 24178.925,E2 24178.925} C_VEL
LIN {X 0,Y 496.978,Z 379.83,A -85,B 0,C 180,E1 24177.457,E2 24177.457} C_VEL
LIN {X 0,Y 496.727,Z 386.989,A -85,B 0,C 180,E1 24175.823,E2 24175.823} C_VEL
LIN {X 0,Y 496.558,Z 392.489,A -85,B 0,C 180,E1 24174.044,E2 24174.044} C_VEL
LIN {X 0,Y 496.466,Z 395.836,A -85,B 0,C 180,E1 24172.325,E2 24172.325} C_VEL
LIN {X 0,Y 496.44,Z 397.447,A -85,B 0,C 180,E1 24170.622,E2 24170.622} C_VEL
LIN {X 0,Y 496.455,Z 397.268,A -85,B 0,C 180,E1 24168.808,E2 24168.808} C_VEL
LIN {X 0,Y 496.528,Z 395.371,A -85,B 0,C 180,E1 24167.107,E2 24167.107} C_VEL
LIN {X 0,Y 496.664,Z 391.621,A -85,B 0,C 180,E1 24165.365,E2 24165.365} C_VEL
LIN {X 0,Y 496.875,Z 385.894,A -85,B 0,C 180,E1 24163.648,E2 24163.648} C_VEL
LIN {X 0,Y 497.174,Z 378.749,A -85,B 0,C 180,E1 24162.09,E2 24162.09} C_VEL
LIN {X 0,Y 497.588,Z 369.64,A -85,B 0,C 180,E1 24160.575,E2 24160.575} C_VEL
LIN {X 0,Y 498.083,Z 358.677,A -85,B 0,C 180,E1 24159.17,E2 24159.17} C_VEL
LIN {X 0,Y 498.583,Z 346.836,A -85,B 0,C 180,E1 24157.989,E2 24157.989} C_VEL
LIN {X 0,Y 499.085,Z 334.154,A -85,B 0,C 180,E1 24157,E2 24157} C_VEL
LIN {X 0,Y 499.551,Z 319.87,A -85,B 0,C 180,E1 24156.154,E2 24156.154} C_VEL
LIN {X 0,Y 499.906,Z 304.685,A -85,B 0,C 180,E1 24155.514,E2 24155.514} C_VEL
LIN {X 0,Y 500.124,Z 289.717,A -85,B 0,C 180,E1 24155.108,E2 24155.108} C_VEL
LIN {X 0,Y 501.243,Z 187.365,A -85,B 0,C 180,E1 24153.429,E2 24153.429} C_VEL
LIN {X 0,Y 498.926,Z 174.449,A -85,B 0,C 180,E1 24153.066,E2 24153.066} C_VEL
LIN {X 0,Y 500.027,Z 145.026,A -85,B 0,C 180,E1 24149.466,E2 24149.466} C_VEL
LIN {X 0,Y 501.342,Z 116.399,A -85,B 0,C 180,E1 24145.898,E2 24145.898} C_VEL
LIN {X 0,Y 502.804,Z 87.171,A -85,B 0,C 180,E1 24142.2,E2 24142.2} C_VEL
LIN {X 0,Y 502.903,Z 81.535,A -85,B 0,C 180,E1 24141.459,E2 24141.459} C_VEL
LIN {X 0,Y 498.183,Z 64.833,A -85,B 0,C 180,E1 24138.853,E2 24138.853} C_VEL
LIN {X 0,Y 496.789,Z 60.039,A -85,B 0,C 180,E1 24138.026,E2 24138.026} C_VEL
LIN {X 0,Y 496.751,Z 59.92,A -85,B 0,C 180,E1 24134.453,E2 24134.453} C_VEL
LIN {X 0,Y 496.723,Z 59.92,A -85,B 0,C 180,E1 24131.025,E2 24131.025} C_VEL
LIN {X 0,Y 496.722,Z 59.923,A -85,B 0,C 180,E1 24127.402,E2 24127.402} C_VEL
LIN {X 0,Y 496.757,Z 59.922,A -85,B 0,C 180,E1 24124.04,E2 24124.04} C_VEL
LIN {X 0,Y 496.77,Z 59.918,A -85,B 0,C 180,E1 24120.462,E2 24120.462} C_VEL
LIN {X 0,Y 496.727,Z 59.921,A -85,B 0,C 180,E1 24117,E2 24117} C_VEL
LIN {X 0,Y 496.712,Z 59.922,A -85,B 0,C 180,E1 24113.528,E2 24113.528} C_VEL
LIN {X 0,Y 496.736,Z 59.922,A -85,B 0,C 180,E1 24110.149,E2 24110.149} C_VEL
LIN {X 0,Y 496.767,Z 59.922,A -85,B 0,C 180,E1 24106.617,E2 24106.617} C_VEL
LIN {X 0,Y 496.729,Z 59.919,A -85,B 0,C 180,E1 24103.151,E2 24103.151} C_VEL
LIN {X 0,Y 496.706,Z 59.921,A -85,B 0,C 180,E1 24099.726,E2 24099.726} C_VEL
